gfCNCPoint2[9660] = {X 255.0630, Y 50.0697, Z -3.0000, A 0.000, B 0.000, C 0.000 }
gfCNCPoint2[9661] = {X 254.3405, Y 49.1989, Z -3.0000, A 0.000, B 0.000, C 0.000 }
gfCNCPoint2[9662] = {X 253.7617, Y 48.2267, Z -3.0000, A 0.000, B 0.000, C 0.000 }
gfCNCPoint2[9663] = {X 253.3406, Y 47.1766, Z -3.0000, A 0.000, B 0.000, C 0.000 }
gfCNCPoint2[9664] = {X 252.9194, Y 48.2267, Z -3.0000, A 0.000, B 0.000, C 0.000 }
gfCNCPoint2[9665] = {X 252.3406, Y 49.1989, Z -3.0000, A 0.000, B 0.000, C 0.000 }
gfCNCPoint2[9666] = {X 251.6182, Y 50.0697, Z -3.0000, A 0.000, B 0.000, C 0.000 }
gfCNCPoint2[9667] = {X 251.5688, Y 50.1201, Z -3.0000, A 0.000, B 0.000, C 0.000 }
gfCNCPoint2[9668] = {X 251.5189, Y 50.1700, Z -3.0000, A 0.000, B 0.000, C 0.000 }
gfCNCPoint2[9669] = {X 250.7133, Y 50.8599, Z -3.0000, A 0.000, B 0.000, C 0.000 }
gfCNCPoint2[9670] = {X 249.8160, Y 51.4254, Z -3.0000, A 0.000, B 0.000, C 0.000 }
gfCNCPoint2[9671] = {X 248.8461, Y 51.8545, Z -3.0000, A 0.000, B 0.000, C 0.000 }
gfCNCPoint2[9672] = {X 247.8241, Y 52.1381, Z -3.0000, A 0.000, B 0.000, C 0.000 }
gfCNCPoint2[9673] = {X 247.8929, Y 52.2639, Z -3.0000, A 0.000, B 0.000, C 0.000 }
gfCNCPoint2[9674] = {X 247.9603, Y 52.3905, Z -3.0000, A 0.000, B 0.000, C 0.000 }
gfCNCPoint2[9675] = {X 250.3409, Y 53.3186, Z -3.0000, A 0.000, B 0.000, C 0.000 }
gfCNCPoint2[9676] = {X 264.1528, Y 58.7989, Z -3.0000, A 0.000, B 0.000, C 0.000 }
gfCNCPoint2[9677] = {X 264.1527, Y 58.0000, Z -3.0000, A 0.000, B 0.000, C 0.000 }
gfCNCPoint2[9678] = {X 264.2034, Y 56.8945, Z -3.0000, A 0.000, B 0.000, C 0.000 }
gfCNCPoint2[9679] = {X 264.3550, Y 55.7982, Z -3.0000, A 0.000, B 0.000, C 0.000 }
gfCNCPoint2[9680] = {X 264.4114, Y 55.5135, Z -3.0000, A 0.000, B 0.000, C 0.000 }
gfCNCPoint2[9681] = {X 264.4745, Y 55.2303, Z -3.0000, A 0.000, B 0.000, C 0.000 }
gfCNCPoint2[9682] = {X 264.9369, Y 53.7185, Z -3.0000, A 0.000, B 0.000, C 0.000 }
gfCNCPoint2[9683] = {X 265.5928, Y 52.2800, Z -3.0000, A 0.000, B 0.000, C 0.000 }
gfCNCPoint2[9684] = {X 262.1384, Y 52.2800, Z -3.0000, A 0.000, B 0.000, C 0.000 }
gfCNCPoint2[9685] = {X 262.1384, Y 49.8800, Z -3.0000, A 0.000, B 0.000, C 0.000 }
gfCNCPoint2[9686] = {X 260.2876, Y 49.8800, Z -3.0000, A 0.000, B 0.000, C 0.000 }
gfCNCPoint2[9687] = {X 259.2646, Y 49.7716, Z -3.0000, A 0.000, B 0.000, C 0.000 }
gfCNCPoint2[9688] = {X 258.2870, Y 49.4511, Z -3.0000, A 0.000, B 0.000, C 0.000 }
gfCNCPoint2[9689] = {X 257.3984, Y 48.9328, Z -3.0000, A 0.000, B 0.000, C 0.000 }
gfCNCPoint2[9690] = {X 256.6382, Y 48.2398, Z -3.0000, A 0.000, B 0.000, C 0.000 }
gfCNCPoint2[9691] = {X 256.0401, Y 47.4028, Z -3.0000, A 0.000, B 0.000, C 0.000 }
gfCNCPoint2[9692] = {X 255.6308, Y 46.4590, Z -3.0000, A 0.000, B 0.000, C 0.000 }
gfCNCPoint2[9693] = {X 255.4666, Y 45.7568, Z -3.0000, A 0.000, B 0.000, C 0.000 }
gfCNCPoint2[9694] = {X 255.4077, Y 45.0380, Z -3.0000, A 0.000, B 0.000, C 0.000 }
gfCNCPoint2[9695] = {X 255.4080, Y 44.1416, Z -3.0000, A 0.000, B 0.000, C 0.000 }
gfCNCPoint2[9696] = {X 255.5183, Y 43.1751, Z -3.0000, A 0.000, B 0.000, C 0.000 }
gfCNCPoint2[9697] = {X 255.8181, Y 42.2496, Z -3.0000, A 0.000, B 0.000, C 0.000 }
gfCNCPoint2[9698] = {X 256.2955, Y 41.4020, Z -3.0000, A 0.000, B 0.000, C 0.000 }
gfCNCPoint2[9699] = {X 256.9315, Y 40.6660, Z -3.0000, A 0.000, B 0.000, C 0.000 }
gfCNCPoint2[9700] = {X 256.9315, Y 35.0338, Z -3.0000, A 0.000, B 0.000, C 0.000 }
gfCNCPoint2[9701] = {X 255.1091, Y 35.0338, Z -3.0000, A 0.000, B 0.000, C 0.000 }
gfCNCPoint2[9702] = {X 251.0864, Y 42.8703, Z -3.0000, A 0.000, B 0.000, C 0.000 }
gfCNCPoint2[9703] = {X 251.2236, Y 43.5126, Z -3.0000, A 0.000, B 0.000, C 0.000 }
gfCNCPoint2[9704] = {X 251.2734, Y 44.1675, Z -3.0000, A 0.000, B 0.000, C 0.000 }
gfCNCPoint2[9705] = {X 251.2736, Y 45.0000, Z -3.0000, A 0.000, B 0.000, C 0.000 }
gfCNCPoint2[9706] = {X 251.2174, Y 45.7380, Z -3.0000, A 0.000, B 0.000, C 0.000 }
gfCNCPoint2[9707] = {X 251.0503, Y 46.4590, Z -3.0000, A 0.000, B 0.000, C 0.000 }
gfCNCPoint2[9708] = {X 250.6346, Y 47.4142, Z -3.0000, A 0.000, B 0.000, C 0.000 }
gfCNCPoint2[9709] = {X 250.0255, Y 48.2593, Z -3.0000, A 0.000, B 0.000, C 0.000 }
gfCNCPoint2[9710] = {X 249.2510, Y 48.9560, Z -3.0000, A 0.000, B 0.000, C 0.000 }
gfCNCPoint2[9711] = {X 248.3462, Y 49.4723, Z -3.0000, A 0.000, B 0.000, C 0.000 }
gfCNCPoint2[9712] = {X 247.3525, Y 49.7849, Z -3.0000, A 0.000, B 0.000, C 0.000 }
gfCNCPoint2[9713] = {X 246.8754, Y 49.8562, Z -3.0000, A 0.000, B 0.000, C 0.000 }
gfCNCPoint2[9714] = {X 246.3936, Y 49.8800, Z -3.0000, A 0.000, B 0.000, C 0.000 }
gfCNCPoint2[9715] = {X 242.5312, Y 49.8800, Z -3.0000, A 0.000, B 0.000, C 0.000 }
gfCNCPoint2[9716] = {X 242.5312, Y 49.4000, Z -3.0000, A 0.000, B 0.000, C 0.000 }
gfCNCPoint2[9717] = {X 239.8075, Y 49.4000, Z -3.0000, A 0.000, B 0.000, C 0.000 }
gfCNCPoint2[9718] = {X 238.8284, Y 49.2897, Z -3.0000, A 0.000, B 0.000, C 0.000 }
gfCNCPoint2[9719] = {X 237.8984, Y 48.9643, Z -3.0000, A 0.000, B 0.000, C 0.000 }
gfCNCPoint2[9720] = {X 237.0641, Y 48.4401, Z -3.0000, A 0.000, B 0.000, C 0.000 }
gfCNCPoint2[9721] = {X 236.3674, Y 47.7434, Z -3.0000, A 0.000, B 0.000, C 0.000 }
gfCNCPoint2[9722] = {X 235.8432, Y 46.9091, Z -3.0000, A 0.000, B 0.000, C 0.000 }
gfCNCPoint2[9723] = {X 235.5178, Y 45.9791, Z -3.0000, A 0.000, B 0.000, C 0.000 }
gfCNCPoint2[9724] = {X 235.4075, Y 45.0000, Z -3.0000, A 0.000, B 0.000, C 0.000 }
gfCNCPoint2[9725] = {X 235.4079, Y 44.1483, Z -3.0000, A 0.000, B 0.000, C 0.000 }
gfCNCPoint2[9726] = {X 235.5063, Y 43.2816, Z -3.0000, A 0.000, B 0.000, C 0.000 }
gfCNCPoint2[9727] = {X 235.7737, Y 42.4514, Z -3.0000, A 0.000, B 0.000, C 0.000 }
gfCNCPoint2[9728] = {X 236.1996, Y 41.6903, Z -3.0000, A 0.000, B 0.000, C 0.000 }
gfCNCPoint2[9729] = {X 236.7672, Y 41.0281, Z -3.0000, A 0.000, B 0.000, C 0.000 }
gfCNCPoint2[9730] = {X 237.4544, Y 40.4909, Z -3.0000, A 0.000, B 0.000, C 0.000 }
gfCNCPoint2[9731] = {X 238.2339, Y 40.0998, Z -3.0000, A 0.000, B 0.000, C 0.000 }
gfCNCPoint2[9732] = {X 242.1750, Y 32.3856, Z -3.0000, A 0.000, B 0.000, C 0.000 }
gfCNCPoint2[9733] = {X 241.0115, Y 31.5932, Z -3.0000, A 0.000, B 0.000, C 0.000 }
gfCNCPoint2[9734] = {X 239.9546, Y 30.6635, Z -3.0000, A 0.000, B 0.000, C 0.000 }
gfCNCPoint2[9735] = {X 239.0203, Y 29.6105, Z -3.0000, A 0.000, B 0.000, C 0.000 }
gfCNCPoint2[9736] = {X 238.2230, Y 28.4504, Z -3.0000, A 0.000, B 0.000, C 0.000 }
gfCNCPoint2[9737] = {X 237.5748, Y 27.2009, Z -3.0000, A 0.000, B 0.000, C 0.000 }
gfCNCPoint2[9738] = {X 237.0856, Y 25.8809, Z -3.0000, A 0.000, B 0.000, C 0.000 }
gfCNCPoint2[9739] = {X 236.6638, Y 24.0613, Z -3.0000, A 0.000, B 0.000, C 0.000 }
gfCNCPoint2[9740] = {X 236.4490, Y 22.2058, Z -3.0000, A 0.000, B 0.000, C 0.000 }
gfCNCPoint2[9741] = {X 236.4438, Y 20.3378, Z -3.0000, A 0.000, B 0.000, C 0.000 }
gfCNCPoint2[9742] = {X 236.6483, Y 18.4812, Z -3.0000, A 0.000, B 0.000, C 0.000 }
gfCNCPoint2[9743] = {X 237.0599, Y 16.6592, Z -3.0000, A 0.000, B 0.000, C 0.000 }
gfCNCPoint2[9744] = {X 237.6340, Y 15.0730, Z -3.0000, A 0.000, B 0.000, C 0.000 }
gfCNCPoint2[9745] = {X 238.4262, Y 13.5836, Z -3.0000, A 0.000, B 0.000, C 0.000 }
gfCNCPoint2[9746] = {X 239.4206, Y 12.2210, Z -3.0000, A 0.000, B 0.000, C 0.000 }
gfCNCPoint2[9747] = {X 240.5972, Y 11.0123, Z -3.0000, A 0.000, B 0.000, C 0.000 }
gfCNCPoint2[9748] = {X 241.9327, Y 9.9816, Z -3.0000, A 0.000, B 0.000, C 0.000 }
gfCNCPoint2[9749] = {X 243.4002, Y 9.1497, Z -3.0000, A 0.000, B 0.000, C 0.000 }
gfCNCPoint2[9750] = {X 244.9704, Y 8.5332, Z -3.0000, A 0.000, B 0.000, C 0.000 }
gfCNCPoint2[9751] = {X 246.6119, Y 8.1444, Z -3.0000, A 0.000, B 0.000, C 0.000 }
gfCNCPoint2[9752] = {X 248.7155, Y 7.8721, Z -3.0000, A 0.000, B 0.000, C 0.000 }
gfCNCPoint2[9753] = {X 250.8351, Y 7.7912, Z -3.0000, A 0.000, B 0.000, C 0.000 }
gfCNCPoint2[9754] = {X 266.7640, Y 7.7912, Z -3.0000, A 0.000, B 0.000, C 0.000 }
gfCNCPoint2[9755] = {X 267.7368, Y 7.9081, Z -3.0000, A 0.000, B 0.000, C 0.000 }
gfCNCPoint2[9756] = {X 268.6596, Y 8.2373, Z -3.0000, A 0.000, B 0.000, C 0.000 }
gfCNCPoint2[9757] = {X 269.4868, Y 8.7623, Z -3.0000, A 0.000, B 0.000, C 0.000 }
gfCNCPoint2[9758] = {X 270.1773, Y 9.4573, Z -3.0000, A 0.000, B 0.000, C 0.000 }
gfCNCPoint2[9759] = {X 270.6971, Y 10.2878, Z -3.0000, A 0.000, B 0.000, C 0.000 }
gfCNCPoint2[9760] = {X 271.0203, Y 11.2127, Z -3.0000, A 0.000, B 0.000, C 0.000 }
gfCNCPoint2[9761] = {X 271.1310, Y 12.1862, Z -3.0000, A 0.000, B 0.000, C 0.000 }
gfCNCPoint2[9762] = {X 271.1308, Y 13.0233, Z -3.0000, A 0.000, B 0.000, C 0.000 }
gfCNCPoint2[9763] = {X 271.0225, Y 13.9494, Z -3.0000, A 0.000, B 0.000, C 0.000 }
gfCNCPoint2[9764] = {X 270.7215, Y 14.8318, Z -3.0000, A 0.000, B 0.000, C 0.000 }
gfCNCPoint2[9765] = {X 270.2413, Y 15.6310, Z -3.0000, A 0.000, B 0.000, C 0.000 }
gfCNCPoint2[9766] = {X 269.6034, Y 16.3111, Z -3.0000, A 0.000, B 0.000, C 0.000 }
gfCNCPoint2[9767] = {X 269.6032, Y 40.8756, Z -3.0000, A 0.000, B 0.000, C 0.000 }
gfCNCPoint2[9768] = {X 270.2480, Y 41.5647, Z -3.0000, A 0.000, B 0.000, C 0.000 }
gfCNCPoint2[9769] = {X 270.7309, Y 42.3755, Z -3.0000, A 0.000, B 0.000, C 0.000 }
gfCNCPoint2[9770] = {X 271.0299, Y 43.2706, Z -3.0000, A 0.000, B 0.000, C 0.000 }
gfCNCPoint2[9771] = {X 271.1310, Y 44.2089, Z -3.0000, A 0.000, B 0.000, C 0.000 }
gfCNCPoint2[9772] = {X 271.1310, Y 45.0000, Z -3.0000, A 0.000, B 0.000, C 0.000 }
gfCNCPoint2[9773] = {X 271.0207, Y 45.9791, Z -3.0000, A 0.000, B 0.000, C 0.000 }
gfCNCPoint2[9774] = {X 270.6953, Y 46.9091, Z -3.0000, A 0.000, B 0.000, C 0.000 }
gfCNCPoint2[9775] = {X 270.1711, Y 47.7434, Z -3.0000, A 0.000, B 0.000, C 0.000 }
gfCNCPoint2[9776] = {X 269.4744, Y 48.4401, Z -3.0000, A 0.000, B 0.000, C 0.000 }
gfCNCPoint2[9777] = {X 268.6401, Y 48.9643, Z -3.0000, A 0.000, B 0.000, C 0.000 }
gfCNCPoint2[9778] = {X 267.7101, Y 49.2897, Z -3.0000, A 0.000, B 0.000, C 0.000 }
gfCNCPoint2[9779] = {X 266.7310, Y 49.4000, Z -3.0000, A 0.000, B 0.000, C 0.000 }
gfCNCPoint2[9780] = {X 260.2876, Y 49.4000, Z -3.0000, A 0.000, B 0.000, C 0.000 }
gfCNCPoint2[9781] = {X 259.3085, Y 49.2897, Z -3.0000, A 0.000, B 0.000, C 0.000 }
gfCNCPoint2[9782] = {X 258.3785, Y 48.9643, Z -3.0000, A 0.000, B 0.000, C 0.000 }
gfCNCPoint2[9783] = {X 257.5442, Y 48.4400, Z -3.0000, A 0.000, B 0.000, C 0.000 }
gfCNCPoint2[9784] = {X 256.8475, Y 47.7433, Z -3.0000, A 0.000, B 0.000, C 0.000 }
gfCNCPoint2[9785] = {X 256.3233, Y 46.9091, Z -3.0000, A 0.000, B 0.000, C 0.000 }
gfCNCPoint2[9786] = {X 255.9979, Y 45.9791, Z -3.0000, A 0.000, B 0.000, C 0.000 }
gfCNCPoint2[9787] = {X 255.8876, Y 45.0000, Z -3.0000, A 0.000, B 0.000, C 0.000 }
gfCNCPoint2[9788] = {X 255.8880, Y 44.1483, Z -3.0000, A 0.000, B 0.000, C 0.000 }
gfCNCPoint2[9789] = {X 255.9984, Y 43.2275, Z -3.0000, A 0.000, B 0.000, C 0.000 }
gfCNCPoint2[9790] = {X 256.2993, Y 42.3503, Z -3.0000, A 0.000, B 0.000, C 0.000 }
gfCNCPoint2[9791] = {X 256.7775, Y 41.5556, Z -3.0000, A 0.000, B 0.000, C 0.000 }
gfCNCPoint2[9792] = {X 257.4115, Y 40.8789, Z -3.0000, A 0.000, B 0.000, C 0.000 }
gfCNCPoint2[9793] = {X 257.4115, Y 34.5538, Z -3.0000, A 0.000, B 0.000, C 0.000 }
gfCNCPoint2[9794] = {X 254.8159, Y 34.5538, Z -3.0000, A 0.000, B 0.000, C 0.000 }
gfCNCPoint2[9795] = {X 250.5702, Y 42.8248, Z -3.0000, A 0.000, B 0.000, C 0.000 }
gfCNCPoint2[9796] = {X 250.7374, Y 43.5079, Z -3.0000, A 0.000, B 0.000, C 0.000 }
gfCNCPoint2[9797] = {X 250.7936, Y 44.2089, Z -3.0000, A 0.000, B 0.000, C 0.000 }
gfCNCPoint2[9798] = {X 250.7936, Y 45.0000, Z -3.0000, A 0.000, B 0.000, C 0.000 }
gfCNCPoint2[9799] = {X 250.6832, Y 45.9791, Z -3.0000, A 0.000, B 0.000, C 0.000 }
gfCNCPoint2[9800] = {X 250.3578, Y 46.9091, Z -3.0000, A 0.000, B 0.000, C 0.000 }
gfCNCPoint2[9801] = {X 249.8336, Y 47.7434, Z -3.0000, A 0.000, B 0.000, C 0.000 }
gfCNCPoint2[9802] = {X 249.1369, Y 48.4401, Z -3.0000, A 0.000, B 0.000, C 0.000 }
gfCNCPoint2[9803] = {X 248.3026, Y 48.9643, Z -3.0000, A 0.000, B 0.000, C 0.000 }
gfCNCPoint2[9804] = {X 247.3727, Y 49.2897, Z -3.0000, A 0.000, B 0.000, C 0.000 }
gfCNCPoint2[9805] = {X 246.3936, Y 49.4000, Z -3.0000, A 0.000, B 0.000, C 0.000 }
gfCNCPoint2[9806] = {X 242.5312, Y 49.4000, Z -3.0000, A 0.000, B 0.000, C 0.000 }
gfCNCPoint2[9807] = {X 242.5312, Y 49.8800, Z -3.0000, A 0.000, B 0.000, C 0.000 }
gfCNCPoint2[9808] = {X 243.4812, Y 50.5824, Z -3.0000, A 0.000, B 0.000, C 0.000 }
gfCNCPoint2[9809] = {X 244.3384, Y 51.3953, Z -3.0000, A 0.000, B 0.000, C 0.000 }
gfCNCPoint2[9810] = {X 245.0903, Y 52.3066, Z -3.0000, A 0.000, B 0.000, C 0.000 }
gfCNCPoint2[9811] = {X 245.7256, Y 53.3027, Z -3.0000, A 0.000, B 0.000, C 0.000 }
gfCNCPoint2[9812] = {X 245.9756, Y 53.7844, Z -3.0000, A 0.000, B 0.000, C 0.000 }
gfCNCPoint2[9813] = {X 246.1981, Y 54.2794, Z -3.0000, A 0.000, B 0.000, C 0.000 }
gfCNCPoint2[9814] = {X 249.4592, Y 55.5508, Z -3.0000, A 0.000, B 0.000, C 0.000 }
gfCNCPoint2[9815] = {X 267.2831, Y 62.6229, Z -3.0000, A 0.000, B 0.000, C 0.000 }
gfCNCPoint2[9816] = {X 266.8847, Y 61.4476, Z -3.0000, A 0.000, B 0.000, C 0.000 }
gfCNCPoint2[9817] = {X 266.6400, Y 60.2310, Z -3.0000, A 0.000, B 0.000, C 0.000 }
gfCNCPoint2[9818] = {X 266.5529, Y 58.9930, Z -3.0000, A 0.000, B 0.000, C 0.000 }
gfCNCPoint2[9819] = {X 266.5527, Y 58.0000, Z -3.0000, A 0.000, B 0.000, C 0.000 }
gfCNCPoint2[9820] = {X 266.6262, Y 56.8093, Z -3.0000, A 0.000, B 0.000, C 0.000 }
gfCNCPoint2[9821] = {X 266.8456, Y 55.6367, Z -3.0000, A 0.000, B 0.000, C 0.000 }
gfCNCPoint2[9822] = {X 267.2076, Y 54.5000, Z -3.0000, A 0.000, B 0.000, C 0.000 }
gfCNCPoint2[9823] = {X 267.7067, Y 53.4164, Z -3.0000, A 0.000, B 0.000, C 0.000 }
gfCNCPoint2[9824] = {X 268.4728, Y 52.2132, Z -3.0000, A 0.000, B 0.000, C 0.000 }
gfCNCPoint2[9825] = {X 269.4075, Y 51.1357, Z -3.0000, A 0.000, B 0.000, C 0.000 }
gfCNCPoint2[9826] = {X 270.4903, Y 50.2072, Z -3.0000, A 0.000, B 0.000, C 0.000 }
gfCNCPoint2[9827] = {X 271.6979, Y 49.4479, Z -3.0000, A 0.000, B 0.000, C 0.000 }
gfCNCPoint2[9828] = {X 273.0039, Y 48.8744, Z -3.0000, A 0.000, B 0.000, C 0.000 }
gfCNCPoint2[9829] = {X 274.3800, Y 48.4989, Z -3.0000, A 0.000, B 0.000, C 0.000 }
gfCNCPoint2[9830] = {X 275.3020, Y 48.3648, Z -3.0000, A 0.000, B 0.000, C 0.000 }
gfCNCPoint2[9831] = {X 276.2327, Y 48.3200, Z -3.0000, A 0.000, B 0.000, C 0.000 }
gfCNCPoint2[9832] = {X 281.0411, Y 48.3200, Z -3.0000, A 0.000, B 0.000, C 0.000 }
gfCNCPoint2[9833] = {X 280.4347, Y 47.5134, Z -3.0000, A 0.000, B 0.000, C 0.000 }
gfCNCPoint2[9834] = {X 280.0072, Y 46.5992, Z -3.0000, A 0.000, B 0.000, C 0.000 }
gfCNCPoint2[9835] = {X 279.7768, Y 45.6167, Z -3.0000, A 0.000, B 0.000, C 0.000 }
gfCNCPoint2[9836] = {X 279.7488, Y 45.3288, Z -3.0000, A 0.000, B 0.000, C 0.000 }
gfCNCPoint2[9837] = {X 279.7378, Y 45.0398, Z -3.0000, A 0.000, B 0.000, C 0.000 }
gfCNCPoint2[9838] = {X 279.7377, Y 44.2039, Z -3.0000, A 0.000, B 0.000, C 0.000 }
gfCNCPoint2[9839] = {X 279.8424, Y 43.2205, Z -3.0000, A 0.000, B 0.000, C 0.000 }
gfCNCPoint2[9840] = {X 280.1412, Y 42.2777, Z -3.0000, A 0.000, B 0.000, C 0.000 }
gfCNCPoint2[9841] = {X 280.6222, Y 41.4136, Z -3.0000, A 0.000, B 0.000, C 0.000 }
gfCNCPoint2[9842] = {X 281.2659, Y 40.6627, Z -3.0000, A 0.000, B 0.000, C 0.000 }
gfCNCPoint2[9843] = {X 281.2655, Y 16.5245, Z -3.0000, A 0.000, B 0.000, C 0.000 }
gfCNCPoint2[9844] = {X 280.6242, Y 15.7828, Z -3.0000, A 0.000, B 0.000, C 0.000 }
gfCNCPoint2[9845] = {X 280.1442, Y 14.9280, Z -3.0000, A 0.000, B 0.000, C 0.000 }
gfCNCPoint2[9846] = {X 279.8447, Y 13.9944, Z -3.0000, A 0.000, B 0.000, C 0.000 }
gfCNCPoint2[9847] = {X 279.7378, Y 13.0198, Z -3.0000, A 0.000, B 0.000, C 0.000 }
gfCNCPoint2[9848] = {X 279.7377, Y 12.1868, Z -3.0000, A 0.000, B 0.000, C 0.000 }
gfCNCPoint2[9849] = {X 279.8242, Y 11.2717, Z -3.0000, A 0.000, B 0.000, C 0.000 }
gfCNCPoint2[9850] = {X 280.0808, Y 10.3891, Z -3.0000, A 0.000, B 0.000, C 0.000 }
gfCNCPoint2[9851] = {X 280.5256, Y 9.5281, Z -3.0000, A 0.000, B 0.000, C 0.000 }
gfCNCPoint2[9852] = {X 281.1317, Y 8.7718, Z -3.0000, A 0.000, B 0.000, C 0.000 }
gfCNCPoint2[9853] = {X 281.8752, Y 8.1503, Z -3.0000, A 0.000, B 0.000, C 0.000 }
gfCNCPoint2[9854] = {X 282.7270, Y 7.6880, Z -3.0000, A 0.000, B 0.000, C 0.000 }
gfCNCPoint2[9855] = {X 283.6533, Y 7.4030, Z -3.0000, A 0.000, B 0.000, C 0.000 }
gfCNCPoint2[9856] = {X 284.6177, Y 7.3068, Z -3.0000, A 0.000, B 0.000, C 0.000 }
gfCNCPoint2[9857] = {X 291.0611, Y 7.3068, Z -3.0000, A 0.000, B 0.000, C 0.000 }
gfCNCPoint2[9858] = {X 292.0255, Y 7.4030, Z -3.0000, A 0.000, B 0.000, C 0.000 }
gfCNCPoint2[9859] = {X 292.9518, Y 7.6880, Z -3.0000, A 0.000, B 0.000, C 0.000 }
gfCNCPoint2[9860] = {X 293.8036, Y 8.1503, Z -3.0000, A 0.000, B 0.000, C 0.000 }
gfCNCPoint2[9861] = {X 294.5471, Y 8.7718, Z -3.0000, A 0.000, B 0.000, C 0.000 }
gfCNCPoint2[9862] = {X 295.1533, Y 9.5281, Z -3.0000, A 0.000, B 0.000, C 0.000 }
gfCNCPoint2[9863] = {X 295.5980, Y 10.3891, Z -3.0000, A 0.000, B 0.000, C 0.000 }
gfCNCPoint2[9864] = {X 295.8044, Y 11.0397, Z -3.0000, A 0.000, B 0.000, C 0.000 }
gfCNCPoint2[9865] = {X 295.9180, Y 11.7127, Z -3.0000, A 0.000, B 0.000, C 0.000 }
gfCNCPoint2[9866] = {X 295.9354, Y 11.9495, Z -3.0000, A 0.000, B 0.000, C 0.000 }
gfCNCPoint2[9867] = {X 295.9411, Y 12.1868, Z -3.0000, A 0.000, B 0.000, C 0.000 }
gfCNCPoint2[9868] = {X 295.9409, Y 13.0237, Z -3.0000, A 0.000, B 0.000, C 0.000 }
gfCNCPoint2[9869] = {X 295.9342, Y 13.2382, Z -3.0000, A 0.000, B 0.000, C 0.000 }
gfCNCPoint2[9870] = {X 295.9180, Y 13.4521, Z -3.0000, A 0.000, B 0.000, C 0.000 }
gfCNCPoint2[9871] = {X 298.3067, Y 13.6853, Z -3.0000, A 0.000, B 0.000, C 0.000 }
gfCNCPoint2[9872] = {X 298.1360, Y 14.6938, Z -3.0000, A 0.000, B 0.000, C 0.000 }
gfCNCPoint2[9873] = {X 297.8257, Y 15.6685, Z -3.0000, A 0.000, B 0.000, C 0.000 }
gfCNCPoint2[9874] = {X 297.3819, Y 16.5900, Z -3.0000, A 0.000, B 0.000, C 0.000 }
gfCNCPoint2[9875] = {X 296.8132, Y 17.4403, Z -3.0000, A 0.000, B 0.000, C 0.000 }
gfCNCPoint2[9876] = {X 296.8136, Y 19.2365, Z -3.0000, A 0.000, B 0.000, C 0.000 }
gfCNCPoint2[9877] = {X 299.7997, Y 19.2365, Z -3.0000, A 0.000, B 0.000, C 0.000 }
gfCNCPoint2[9878] = {X 299.7999, Y 17.4399, Z -3.0000, A 0.000, B 0.000, C 0.000 }
gfCNCPoint2[9879] = {X 299.2314, Y 16.5898, Z -3.0000, A 0.000, B 0.000, C 0.000 }
gfCNCPoint2[9880] = {X 298.7876, Y 15.6683, Z -3.0000, A 0.000, B 0.000, C 0.000 }
gfCNCPoint2[9881] = {X 298.4773, Y 14.6937, Z -3.0000, A 0.000, B 0.000, C 0.000 }
gfCNCPoint2[9882] = {X 298.3067, Y 13.6853, Z -3.0000, A 0.000, B 0.000, C 0.000 }
gfCNCPoint2[9883] = {X 295.9180, Y 13.4521, Z -3.0000, A 0.000, B 0.000, C 0.000 }
gfCNCPoint2[9884] = {X 295.7559, Y 14.3097, Z -3.0000, A 0.000, B 0.000, C 0.000 }
gfCNCPoint2[9885] = {X 295.4436, Y 15.1246, Z -3.0000, A 0.000, B 0.000, C 0.000 }
gfCNCPoint2[9886] = {X 294.9912, Y 15.8710, Z -3.0000, A 0.000, B 0.000, C 0.000 }
gfCNCPoint2[9887] = {X 294.4130, Y 16.5247, Z -3.0000, A 0.000, B 0.000, C 0.000 }
gfCNCPoint2[9888] = {X 294.4141, Y 21.6365, Z -3.0000, A 0.000, B 0.000, C 0.000 }
gfCNCPoint2[9889] = {X 302.1995, Y 21.6365, Z -3.0000, A 0.000, B 0.000, C 0.000 }
gfCNCPoint2[9890] = {X 302.2000, Y 16.5244, Z -3.0000, A 0.000, B 0.000, C 0.000 }
gfCNCPoint2[9891] = {X 301.6220, Y 15.8706, Z -3.0000, A 0.000, B 0.000, C 0.000 }
gfCNCPoint2[9892] = {X 301.1696, Y 15.1244, Z -3.0000, A 0.000, B 0.000, C 0.000 }
gfCNCPoint2[9893] = {X 300.8574, Y 14.3095, Z -3.0000, A 0.000, B 0.000, C 0.000 }
gfCNCPoint2[9894] = {X 300.6953, Y 13.4521, Z -3.0000, A 0.000, B 0.000, C 0.000 }
gfCNCPoint2[9895] = {X 300.6791, Y 13.2371, Z -3.0000, A 0.000, B 0.000, C 0.000 }
gfCNCPoint2[9896] = {X 300.6724, Y 13.0215, Z -3.0000, A 0.000, B 0.000, C 0.000 }
gfCNCPoint2[9897] = {X 300.6723, Y 12.1868, Z -3.0000, A 0.000, B 0.000, C 0.000 }
gfCNCPoint2[9898] = {X 300.6780, Y 11.9495, Z -3.0000, A 0.000, B 0.000, C 0.000 }
gfCNCPoint2[9899] = {X 300.6953, Y 11.7127, Z -3.0000, A 0.000, B 0.000, C 0.000 }
gfCNCPoint2[9900] = {X 300.8090, Y 11.0397, Z -3.0000, A 0.000, B 0.000, C 0.000 }
gfCNCPoint2[9901] = {X 301.0154, Y 10.3891, Z -3.0000, A 0.000, B 0.000, C 0.000 }
gfCNCPoint2[9902] = {X 301.4601, Y 9.5281, Z -3.0000, A 0.000, B 0.000, C 0.000 }
gfCNCPoint2[9903] = {X 302.0662, Y 8.7718, Z -3.0000, A 0.000, B 0.000, C 0.000 }
gfCNCPoint2[9904] = {X 302.8098, Y 8.1503, Z -3.0000, A 0.000, B 0.000, C 0.000 }
gfCNCPoint2[9905] = {X 303.6616, Y 7.6880, Z -3.0000, A 0.000, B 0.000, C 0.000 }
gfCNCPoint2[9906] = {X 304.5879, Y 7.4030, Z -3.0000, A 0.000, B 0.000, C 0.000 }
gfCNCPoint2[9907] = {X 305.5523, Y 7.3068, Z -3.0000, A 0.000, B 0.000, C 0.000 }
gfCNCPoint2[9908] = {X 311.9957, Y 7.3068, Z -3.0000, A 0.000, B 0.000, C 0.000 }
gfCNCPoint2[9909] = {X 312.9478, Y 7.4006, Z -3.0000, A 0.000, B 0.000, C 0.000 }
gfCNCPoint2[9910] = {X 313.8632, Y 7.6783, Z -3.0000, A 0.000, B 0.000, C 0.000 }
gfCNCPoint2[9911] = {X 314.7069, Y 8.1292, Z -3.0000, A 0.000, B 0.000, C 0.000 }
gfCNCPoint2[9912] = {X 315.4464, Y 8.7361, Z -3.0000, A 0.000, B 0.000, C 0.000 }
gfCNCPoint2[9913] = {X 316.0533, Y 9.4756, Z -3.0000, A 0.000, B 0.000, C 0.000 }
gfCNCPoint2[9914] = {X 316.5043, Y 10.3193, Z -3.0000, A 0.000, B 0.000, C 0.000 }
gfCNCPoint2[9915] = {X 316.7820, Y 11.2348, Z -3.0000, A 0.000, B 0.000, C 0.000 }
gfCNCPoint2[9916] = {X 316.8757, Y 12.1868, Z -3.0000, A 0.000, B 0.000, C 0.000 }
gfCNCPoint2[9917] = {X 316.8755, Y 13.0237, Z -3.0000, A 0.000, B 0.000, C 0.000 }
gfCNCPoint2[9918] = {X 316.7681, Y 13.9973, Z -3.0000, A 0.000, B 0.000, C 0.000 }
gfCNCPoint2[9919] = {X 316.4684, Y 14.9299, Z -3.0000, A 0.000, B 0.000, C 0.000 }
gfCNCPoint2[9920] = {X 315.9885, Y 15.7838, Z -3.0000, A 0.000, B 0.000, C 0.000 }
gfCNCPoint2[9921] = {X 315.3477, Y 16.5246, Z -3.0000, A 0.000, B 0.000, C 0.000 }
gfCNCPoint2[9922] = {X 315.3475, Y 40.6620, Z -3.0000, A 0.000, B 0.000, C 0.000 }
gfCNCPoint2[9923] = {X 315.9888, Y 41.4035, Z -3.0000, A 0.000, B 0.000, C 0.000 }
gfCNCPoint2[9924] = {X 316.4690, Y 42.2583, Z -3.0000, A 0.000, B 0.000, C 0.000 }
gfCNCPoint2[9925] = {X 316.7686, Y 43.1918, Z -3.0000, A 0.000, B 0.000, C 0.000 }
gfCNCPoint2[9926] = {X 316.8755, Y 44.1664, Z -3.0000, A 0.000, B 0.000, C 0.000 }
gfCNCPoint2[9927] = {X 316.8757, Y 45.0000, Z -3.0000, A 0.000, B 0.000, C 0.000 }
gfCNCPoint2[9928] = {X 316.8749, Y 45.0899, Z -3.0000, A 0.000, B 0.000, C 0.000 }
gfCNCPoint2[9929] = {X 316.8724, Y 45.1799, Z -3.0000, A 0.000, B 0.000, C 0.000 }
gfCNCPoint2[9930] = {X 316.8594, Y 45.3987, Z -3.0000, A 0.000, B 0.000, C 0.000 }
gfCNCPoint2[9931] = {X 316.8366, Y 45.6167, Z -3.0000, A 0.000, B 0.000, C 0.000 }
gfCNCPoint2[9932] = {X 316.6062, Y 46.5992, Z -3.0000, A 0.000, B 0.000, C 0.000 }
gfCNCPoint2[9933] = {X 316.1787, Y 47.5134, Z -3.0000, A 0.000, B 0.000, C 0.000 }
gfCNCPoint2[9934] = {X 315.5723, Y 48.3200, Z -3.0000, A 0.000, B 0.000, C 0.000 }
gfCNCPoint2[9935] = {X 315.2205, Y 47.9934, Z -3.0000, A 0.000, B 0.000, C 0.000 }
gfCNCPoint2[9936] = {X 314.5413, Y 48.5889, Z -3.0000, A 0.000, B 0.000, C 0.000 }
gfCNCPoint2[9937] = {X 313.7548, Y 49.0331, Z -3.0000, A 0.000, B 0.000, C 0.000 }
gfCNCPoint2[9938] = {X 312.8942, Y 49.3073, Z -3.0000, A 0.000, B 0.000, C 0.000 }
gfCNCPoint2[9939] = {X 311.9957, Y 49.4000, Z -3.0000, A 0.000, B 0.000, C 0.000 }
gfCNCPoint2[9940] = {X 305.5523, Y 49.4000, Z -3.0000, A 0.000, B 0.000, C 0.000 }
gfCNCPoint2[9941] = {X 304.5732, Y 49.2897, Z -3.0000, A 0.000, B 0.000, C 0.000 }
gfCNCPoint2[9942] = {X 303.6432, Y 48.9643, Z -3.0000, A 0.000, B 0.000, C 0.000 }
gfCNCPoint2[9943] = {X 302.8089, Y 48.4400, Z -3.0000, A 0.000, B 0.000, C 0.000 }
gfCNCPoint2[9944] = {X 302.1122, Y 47.7433, Z -3.0000, A 0.000, B 0.000, C 0.000 }
gfCNCPoint2[9945] = {X 301.5880, Y 46.9091, Z -3.0000, A 0.000, B 0.000, C 0.000 }
gfCNCPoint2[9946] = {X 301.2626, Y 45.9791, Z -3.0000, A 0.000, B 0.000, C 0.000 }
gfCNCPoint2[9947] = {X 301.1523, Y 45.0000, Z -3.0000, A 0.000, B 0.000, C 0.000 }
gfCNCPoint2[9948] = {X 301.1524, Y 44.1992, Z -3.0000, A 0.000, B 0.000, C 0.000 }
gfCNCPoint2[9949] = {X 301.2703, Y 43.2558, Z -3.0000, A 0.000, B 0.000, C 0.000 }
gfCNCPoint2[9950] = {X 301.5735, Y 42.3546, Z -3.0000, A 0.000, B 0.000, C 0.000 }
gfCNCPoint2[9951] = {X 302.0499, Y 41.5318, Z -3.0000, A 0.000, B 0.000, C 0.000 }
gfCNCPoint2[9952] = {X 302.6804, Y 40.8202, Z -3.0000, A 0.000, B 0.000, C 0.000 }
gfCNCPoint2[9953] = {X 302.6804, Y 34.1143, Z -3.0000, A 0.000, B 0.000, C 0.000 }
gfCNCPoint2[9954] = {X 293.9340, Y 34.1143, Z -3.0000, A 0.000, B 0.000, C 0.000 }
gfCNCPoint2[9955] = {X 293.9331, Y 40.8663, Z -3.0000, A 0.000, B 0.000, C 0.000 }
gfCNCPoint2[9956] = {X 294.5730, Y 41.5612, Z -3.0000, A 0.000, B 0.000, C 0.000 }
gfCNCPoint2[9957] = {X 295.0538, Y 42.3745, Z -3.0000, A 0.000, B 0.000, C 0.000 }
gfCNCPoint2[9958] = {X 295.3543, Y 43.2702, Z -3.0000, A 0.000, B 0.000, C 0.000 }
gfCNCPoint2[9959] = {X 295.4611, Y 44.2089, Z -3.0000, A 0.000, B 0.000, C 0.000 }
gfCNCPoint2[9960] = {X 295.4611, Y 45.0000, Z -3.0000, A 0.000, B 0.000, C 0.000 }
gfCNCPoint2[9961] = {X 295.3508, Y 45.9791, Z -3.0000, A 0.000, B 0.000, C 0.000 }
gfCNCPoint2[9962] = {X 295.0254, Y 46.9091, Z -3.0000, A 0.000, B 0.000, C 0.000 }
gfCNCPoint2[9963] = {X 294.5012, Y 47.7434, Z -3.0000, A 0.000, B 0.000, C 0.000 }
gfCNCPoint2[9964] = {X 293.8045, Y 48.4401, Z -3.0000, A 0.000, B 0.000, C 0.000 }
gfCNCPoint2[9965] = {X 292.9702, Y 48.9643, Z -3.0000, A 0.000, B 0.000, C 0.000 }
gfCNCPoint2[9966] = {X 292.0402, Y 49.2897, Z -3.0000, A 0.000, B 0.000, C 0.000 }
gfCNCPoint2[9967] = {X 291.0611, Y 49.4000, Z -3.0000, A 0.000, B 0.000, C 0.000 }
gfCNCPoint2[9968] = {X 284.6177, Y 49.4000, Z -3.0000, A 0.000, B 0.000, C 0.000 }
gfCNCPoint2[9969] = {X 283.6386, Y 49.2897, Z -3.0000, A 0.000, B 0.000, C 0.000 }
gfCNCPoint2[9970] = {X 282.7086, Y 48.9643, Z -3.0000, A 0.000, B 0.000, C 0.000 }
gfCNCPoint2[9971] = {X 281.8743, Y 48.4400, Z -3.0000, A 0.000, B 0.000, C 0.000 }
gfCNCPoint2[9972] = {X 281.1776, Y 47.7433, Z -3.0000, A 0.000, B 0.000, C 0.000 }
gfCNCPoint2[9973] = {X 280.6534, Y 46.9091, Z -3.0000, A 0.000, B 0.000, C 0.000 }
gfCNCPoint2[9974] = {X 280.3280, Y 45.9791, Z -3.0000, A 0.000, B 0.000, C 0.000 }
gfCNCPoint2[9975] = {X 280.2177, Y 45.0000, Z -3.0000, A 0.000, B 0.000, C 0.000 }
gfCNCPoint2[9976] = {X 280.2177, Y 44.2066, Z -3.0000, A 0.000, B 0.000, C 0.000 }
gfCNCPoint2[9977] = {X 280.3228, Y 43.2697, Z -3.0000, A 0.000, B 0.000, C 0.000 }
gfCNCPoint2[9978] = {X 280.6229, Y 42.3760, Z -3.0000, A 0.000, B 0.000, C 0.000 }
gfCNCPoint2[9979] = {X 281.1045, Y 41.5655, Z -3.0000, A 0.000, B 0.000, C 0.000 }
gfCNCPoint2[9980] = {X 281.7459, Y 40.8746, Z -3.0000, A 0.000, B 0.000, C 0.000 }
gfCNCPoint2[9981] = {X 281.7455, Y 16.3113, Z -3.0000, A 0.000, B 0.000, C 0.000 }
gfCNCPoint2[9982] = {X 281.1008, Y 15.6221, Z -3.0000, A 0.000, B 0.000, C 0.000 }
gfCNCPoint2[9983] = {X 280.6178, Y 14.8114, Z -3.0000, A 0.000, B 0.000, C 0.000 }
gfCNCPoint2[9984] = {X 280.3189, Y 13.9162, Z -3.0000, A 0.000, B 0.000, C 0.000 }
gfCNCPoint2[9985] = {X 280.2177, Y 12.9779, Z -3.0000, A 0.000, B 0.000, C 0.000 }
gfCNCPoint2[9986] = {X 280.2177, Y 12.1868, Z -3.0000, A 0.000, B 0.000, C 0.000 }
gfCNCPoint2[9987] = {X 280.3280, Y 11.2077, Z -3.0000, A 0.000, B 0.000, C 0.000 }
gfCNCPoint2[9988] = {X 280.6534, Y 10.2777, Z -3.0000, A 0.000, B 0.000, C 0.000 }
gfCNCPoint2[9989] = {X 281.1776, Y 9.4435, Z -3.0000, A 0.000, B 0.000, C 0.000 }
gfCNCPoint2[9990] = {X 281.8743, Y 8.7468, Z -3.0000, A 0.000, B 0.000, C 0.000 }
gfCNCPoint2[9991] = {X 282.7086, Y 8.2226, Z -3.0000, A 0.000, B 0.000, C 0.000 }
gfCNCPoint2[9992] = {X 283.6386, Y 7.8971, Z -3.0000, A 0.000, B 0.000, C 0.000 }
gfCNCPoint2[9993] = {X 284.6177, Y 7.7868, Z -3.0000, A 0.000, B 0.000, C 0.000 }
gfCNCPoint2[9994] = {X 291.0611, Y 7.7868, Z -3.0000, A 0.000, B 0.000, C 0.000 }
gfCNCPoint2[9995] = {X 292.0402, Y 7.8971, Z -3.0000, A 0.000, B 0.000, C 0.000 }
gfCNCPoint2[9996] = {X 292.9702, Y 8.2226, Z -3.0000, A 0.000, B 0.000, C 0.000 }
gfCNCPoint2[9997] = {X 293.8045, Y 8.7468, Z -3.0000, A 0.000, B 0.000, C 0.000 }
gfCNCPoint2[9998] = {X 294.5012, Y 9.4435, Z -3.0000, A 0.000, B 0.000, C 0.000 }
gfCNCPoint2[9999] = {X 295.0254, Y 10.2777, Z -3.0000, A 0.000, B 0.000, C 0.000 }
gfCNCPoint2[10000] = {X 295.3508, Y 11.2077, Z -3.0000, A 0.000, B 0.000, C 0.000 }
gfCNCPoint2[10001] = {X 295.4611, Y 12.1868, Z -3.0000, A 0.000, B 0.000, C 0.000 }
gfCNCPoint2[10002] = {X 295.4609, Y 13.0233, Z -3.0000, A 0.000, B 0.000, C 0.000 }
gfCNCPoint2[10003] = {X 295.3525, Y 13.9495, Z -3.0000, A 0.000, B 0.000, C 0.000 }
gfCNCPoint2[10004] = {X 295.0514, Y 14.8321, Z -3.0000, A 0.000, B 0.000, C 0.000 }
gfCNCPoint2[10005] = {X 294.5710, Y 15.6314, Z -3.0000, A 0.000, B 0.000, C 0.000 }
gfCNCPoint2[10006] = {X 293.9330, Y 16.3116, Z -3.0000, A 0.000, B 0.000, C 0.000 }
gfCNCPoint2[10007] = {X 293.9342, Y 22.1165, Z -3.0000, A 0.000, B 0.000, C 0.000 }
gfCNCPoint2[10008] = {X 302.6795, Y 22.1165, Z -3.0000, A 0.000, B 0.000, C 0.000 }
gfCNCPoint2[10009] = {X 302.6800, Y 16.3112, Z -3.0000, A 0.000, B 0.000, C 0.000 }
gfCNCPoint2[10010] = {X 302.0353, Y 15.6221, Z -3.0000, A 0.000, B 0.000, C 0.000 }
gfCNCPoint2[10011] = {X 301.5524, Y 14.8113, Z -3.0000, A 0.000, B 0.000, C 0.000 }
gfCNCPoint2[10012] = {X 301.2534, Y 13.9162, Z -3.0000, A 0.000, B 0.000, C 0.000 }
gfCNCPoint2[10013] = {X 301.1523, Y 12.9779, Z -3.0000, A 0.000, B 0.000, C 0.000 }
gfCNCPoint2[10014] = {X 301.1523, Y 12.1868, Z -3.0000, A 0.000, B 0.000, C 0.000 }
gfCNCPoint2[10015] = {X 301.2626, Y 11.2077, Z -3.0000, A 0.000, B 0.000, C 0.000 }
gfCNCPoint2[10016] = {X 301.5880, Y 10.2777, Z -3.0000, A 0.000, B 0.000, C 0.000 }
gfCNCPoint2[10017] = {X 302.1122, Y 9.4435, Z -3.0000, A 0.000, B 0.000, C 0.000 }
gfCNCPoint2[10018] = {X 302.8089, Y 8.7468, Z -3.0000, A 0.000, B 0.000, C 0.000 }
gfCNCPoint2[10019] = {X 303.6432, Y 8.2226, Z -3.0000, A 0.000, B 0.000, C 0.000 }
gfCNCPoint2[10020] = {X 304.5732, Y 7.8971, Z -3.0000, A 0.000, B 0.000, C 0.000 }
gfCNCPoint2[10021] = {X 305.5523, Y 7.7868, Z -3.0000, A 0.000, B 0.000, C 0.000 }
gfCNCPoint2[10022] = {X 311.9957, Y 7.7868, Z -3.0000, A 0.000, B 0.000, C 0.000 }
gfCNCPoint2[10023] = {X 312.9748, Y 7.8971, Z -3.0000, A 0.000, B 0.000, C 0.000 }
gfCNCPoint2[10024] = {X 313.9048, Y 8.2226, Z -3.0000, A 0.000, B 0.000, C 0.000 }
gfCNCPoint2[10025] = {X 314.7391, Y 8.7468, Z -3.0000, A 0.000, B 0.000, C 0.000 }
gfCNCPoint2[10026] = {X 315.4358, Y 9.4435, Z -3.0000, A 0.000, B 0.000, C 0.000 }
gfCNCPoint2[10027] = {X 315.9600, Y 10.2777, Z -3.0000, A 0.000, B 0.000, C 0.000 }
gfCNCPoint2[10028] = {X 316.2854, Y 11.2077, Z -3.0000, A 0.000, B 0.000, C 0.000 }
gfCNCPoint2[10029] = {X 316.3957, Y 12.1868, Z -3.0000, A 0.000, B 0.000, C 0.000 }
gfCNCPoint2[10030] = {X 316.3955, Y 13.0233, Z -3.0000, A 0.000, B 0.000, C 0.000 }
gfCNCPoint2[10031] = {X 316.2871, Y 13.9495, Z -3.0000, A 0.000, B 0.000, C 0.000 }
gfCNCPoint2[10032] = {X 315.9860, Y 14.8320, Z -3.0000, A 0.000, B 0.000, C 0.000 }
gfCNCPoint2[10033] = {X 315.5057, Y 15.6313, Z -3.0000, A 0.000, B 0.000, C 0.000 }
gfCNCPoint2[10034] = {X 314.8677, Y 16.3114, Z -3.0000, A 0.000, B 0.000, C 0.000 }
gfCNCPoint2[10035] = {X 314.8675, Y 40.8752, Z -3.0000, A 0.000, B 0.000, C 0.000 }
gfCNCPoint2[10036] = {X 315.5124, Y 41.5644, Z -3.0000, A 0.000, B 0.000, C 0.000 }
gfCNCPoint2[10037] = {X 315.9955, Y 42.3752, Z -3.0000, A 0.000, B 0.000, C 0.000 }
gfCNCPoint2[10038] = {X 316.2945, Y 43.2705, Z -3.0000, A 0.000, B 0.000, C 0.000 }
gfCNCPoint2[10039] = {X 316.3957, Y 44.2089, Z -3.0000, A 0.000, B 0.000, C 0.000 }
gfCNCPoint2[10040] = {X 316.3957, Y 45.0000, Z -3.0000, A 0.000, B 0.000, C 0.000 }
gfCNCPoint2[10041] = {X 316.3190, Y 45.8182, Z -3.0000, A 0.000, B 0.000, C 0.000 }
gfCNCPoint2[10042] = {X 316.0914, Y 46.6079, Z -3.0000, A 0.000, B 0.000, C 0.000 }
gfCNCPoint2[10043] = {X 315.7209, Y 47.3415, Z -3.0000, A 0.000, B 0.000, C 0.000 }
gfCNCPoint2[10044] = {X 315.2205, Y 47.9934, Z -3.0000, A 0.000, B 0.000, C 0.000 }
gfCNCPoint2[10045] = {X 315.5723, Y 48.3200, Z -3.0000, A 0.000, B 0.000, C 0.000 }
gfCNCPoint2[10046] = {X 324.3107, Y 48.3200, Z -3.0000, A 0.000, B 0.000, C 0.000 }
gfCNCPoint2[10047] = {X 325.5555, Y 48.4004, Z -3.0000, A 0.000, B 0.000, C 0.000 }
gfCNCPoint2[10048] = {X 326.7797, Y 48.6402, Z -3.0000, A 0.000, B 0.000, C 0.000 }
gfCNCPoint2[10049] = {X 325.5882, Y 48.0963, Z -3.0000, A 0.000, B 0.000, C 0.000 }
gfCNCPoint2[10050] = {X 324.4810, Y 47.3966, Z -3.0000, A 0.000, B 0.000, C 0.000 }
gfCNCPoint2[10051] = {X 323.4784, Y 46.5538, Z -3.0000, A 0.000, B 0.000, C 0.000 }
gfCNCPoint2[10052] = {X 322.8382, Y 45.9295, Z -3.0000, A 0.000, B 0.000, C 0.000 }
gfCNCPoint2[10053] = {X 322.2180, Y 45.2650, Z -3.0000, A 0.000, B 0.000, C 0.000 }
gfCNCPoint2[10054] = {X 321.6628, Y 44.5452, Z -3.0000, A 0.000, B 0.000, C 0.000 }
gfCNCPoint2[10055] = {X 323.6300, Y 43.1703, Z -3.0000, A 0.000, B 0.000, C 0.000 }
gfCNCPoint2[10056] = {X 323.0063, Y 42.0918, Z -3.0000, A 0.000, B 0.000, C 0.000 }
gfCNCPoint2[10057] = {X 322.5757, Y 40.9227, Z -3.0000, A 0.000, B 0.000, C 0.000 }
gfCNCPoint2[10058] = {X 322.3506, Y 39.6973, Z -3.0000, A 0.000, B 0.000, C 0.000 }
gfCNCPoint2[10059] = {X 322.3379, Y 38.4514, Z -3.0000, A 0.000, B 0.000, C 0.000 }
gfCNCPoint2[10060] = {X 322.5377, Y 37.2217, Z -3.0000, A 0.000, B 0.000, C 0.000 }
gfCNCPoint2[10061] = {X 322.9443, Y 36.0440, Z -3.0000, A 0.000, B 0.000, C 0.000 }
gfCNCPoint2[10062] = {X 323.5458, Y 34.9529, Z -3.0000, A 0.000, B 0.000, C 0.000 }
gfCNCPoint2[10063] = {X 327.7790, Y 28.6234, Z -3.0000, A 0.000, B 0.000, C 0.000 }
gfCNCPoint2[10064] = {X 328.5158, Y 27.6951, Z -3.0000, A 0.000, B 0.000, C 0.000 }
gfCNCPoint2[10065] = {X 329.3936, Y 26.8986, Z -3.0000, A 0.000, B 0.000, C 0.000 }
gfCNCPoint2[10066] = {X 330.3889, Y 26.2552, Z -3.0000, A 0.000, B 0.000, C 0.000 }
gfCNCPoint2[10067] = {X 331.5063, Y 25.7713, Z -3.0000, A 0.000, B 0.000, C 0.000 }
gfCNCPoint2[10068] = {X 332.6887, Y 25.4804, Z -3.0000, A 0.000, B 0.000, C 0.000 }
gfCNCPoint2[10069] = {X 333.9031, Y 25.3907, Z -3.0000, A 0.000, B 0.000, C 0.000 }
gfCNCPoint2[10070] = {X 335.1154, Y 25.5046, Z -3.0000, A 0.000, B 0.000, C 0.000 }
gfCNCPoint2[10071] = {X 336.2918, Y 25.8191, Z -3.0000, A 0.000, B 0.000, C 0.000 }
gfCNCPoint2[10072] = {X 337.3993, Y 26.3252, Z -3.0000, A 0.000, B 0.000, C 0.000 }
gfCNCPoint2[10073] = {X 338.1754, Y 26.8291, Z -3.0000, A 0.000, B 0.000, C 0.000 }
gfCNCPoint2[10074] = {X 338.8813, Y 27.4275, Z -3.0000, A 0.000, B 0.000, C 0.000 }
gfCNCPoint2[10075] = {X 339.4514, Y 27.9767, Z -3.0000, A 0.000, B 0.000, C 0.000 }
gfCNCPoint2[10076] = {X 339.8232, Y 28.3622, Z -3.0000, A 0.000, B 0.000, C 0.000 }
gfCNCPoint2[10077] = {X 340.1656, Y 28.7740, Z -3.0000, A 0.000, B 0.000, C 0.000 }
gfCNCPoint2[10078] = {X 345.8671, Y 24.3770, Z -3.0000, A 0.000, B 0.000, C 0.000 }
gfCNCPoint2[10079] = {X 346.4661, Y 25.2135, Z -3.0000, A 0.000, B 0.000, C 0.000 }
gfCNCPoint2[10080] = {X 347.0041, Y 26.0905, Z -3.0000, A 0.000, B 0.000, C 0.000 }
gfCNCPoint2[10081] = {X 347.1181, Y 24.7344, Z -3.0000, A 0.000, B 0.000, C 0.000 }
gfCNCPoint2[10082] = {X 346.9942, Y 23.3793, Z -3.0000, A 0.000, B 0.000, C 0.000 }
gfCNCPoint2[10083] = {X 346.9501, Y 23.1695, Z -3.0000, A 0.000, B 0.000, C 0.000 }
gfCNCPoint2[10084] = {X 346.8820, Y 22.9664, Z -3.0000, A 0.000, B 0.000, C 0.000 }
gfCNCPoint2[10085] = {X 346.3957, Y 23.6869, Z -3.0000, A 0.000, B 0.000, C 0.000 }
gfCNCPoint2[10086] = {X 345.8671, Y 24.3770, Z -3.0000, A 0.000, B 0.000, C 0.000 }
gfCNCPoint2[10087] = {X 343.9666, Y 25.8427, Z -3.0000, A 0.000, B 0.000, C 0.000 }
gfCNCPoint2[10088] = {X 344.4663, Y 26.5405, Z -3.0000, A 0.000, B 0.000, C 0.000 }
gfCNCPoint2[10089] = {X 344.9152, Y 27.2721, Z -3.0000, A 0.000, B 0.000, C 0.000 }
gfCNCPoint2[10090] = {X 345.4669, Y 28.3755, Z -3.0000, A 0.000, B 0.000, C 0.000 }
gfCNCPoint2[10091] = {X 345.9033, Y 29.5293, Z -3.0000, A 0.000, B 0.000, C 0.000 }
gfCNCPoint2[10092] = {X 346.4600, Y 29.6320, Z -3.0000, A 0.000, B 0.000, C 0.000 }
gfCNCPoint2[10093] = {X 347.0261, Y 29.6228, Z -3.0000, A 0.000, B 0.000, C 0.000 }
gfCNCPoint2[10094] = {X 347.4357, Y 29.5576, Z -3.0000, A 0.000, B 0.000, C 0.000 }
gfCNCPoint2[10095] = {X 347.7945, Y 29.3497, Z -3.0000, A 0.000, B 0.000, C 0.000 }
gfCNCPoint2[10096] = {X 348.4751, Y 28.6299, Z -3.0000, A 0.000, B 0.000, C 0.000 }
gfCNCPoint2[10097] = {X 348.9860, Y 27.7811, Z -3.0000, A 0.000, B 0.000, C 0.000 }
gfCNCPoint2[10098] = {X 349.3035, Y 26.8428, Z -3.0000, A 0.000, B 0.000, C 0.000 }
gfCNCPoint2[10099] = {X 349.3377, Y 26.6716, Z -3.0000, A 0.000, B 0.000, C 0.000 }
gfCNCPoint2[10100] = {X 349.3689, Y 26.4998, Z -3.0000, A 0.000, B 0.000, C 0.000 }
gfCNCPoint2[10101] = {X 349.5024, Y 25.3283, Z -3.0000, A 0.000, B 0.000, C 0.000 }
gfCNCPoint2[10102] = {X 349.4996, Y 24.1493, Z -3.0000, A 0.000, B 0.000, C 0.000 }
gfCNCPoint2[10103] = {X 349.3605, Y 22.9785, Z -3.0000, A 0.000, B 0.000, C 0.000 }
gfCNCPoint2[10104] = {X 349.1887, Y 22.2867, Z -3.0000, A 0.000, B 0.000, C 0.000 }
gfCNCPoint2[10105] = {X 348.9033, Y 21.6336, Z -3.0000, A 0.000, B 0.000, C 0.000 }
gfCNCPoint2[10106] = {X 348.5126, Y 21.0375, Z -3.0000, A 0.000, B 0.000, C 0.000 }
gfCNCPoint2[10107] = {X 348.1201, Y 20.6782, Z -3.0000, A 0.000, B 0.000, C 0.000 }
gfCNCPoint2[10108] = {X 347.6259, Y 20.4810, Z -3.0000, A 0.000, B 0.000, C 0.000 }
gfCNCPoint2[10109] = {X 346.5728, Y 20.3825, Z -3.0000, A 0.000, B 0.000, C 0.000 }
gfCNCPoint2[10110] = {X 345.5200, Y 20.4828, Z -3.0000, A 0.000, B 0.000, C 0.000 }
gfCNCPoint2[10111] = {X 344.7178, Y 21.8936, Z -3.0000, A 0.000, B 0.000, C 0.000 }
gfCNCPoint2[10112] = {X 343.7338, Y 23.1841, Z -3.0000, A 0.000, B 0.000, C 0.000 }
gfCNCPoint2[10113] = {X 342.5857, Y 24.3311, Z -3.0000, A 0.000, B 0.000, C 0.000 }
gfCNCPoint2[10114] = {X 342.7815, Y 24.5198, Z -3.0000, A 0.000, B 0.000, C 0.000 }
gfCNCPoint2[10115] = {X 343.3984, Y 25.1594, Z -3.0000, A 0.000, B 0.000, C 0.000 }
gfCNCPoint2[10116] = {X 343.9666, Y 25.8427, Z -3.0000, A 0.000, B 0.000, C 0.000 }
gfCNCPoint2[10117] = {X 342.0661, Y 27.3083, Z -3.0000, A 0.000, B 0.000, C 0.000 }
gfCNCPoint2[10118] = {X 342.8614, Y 28.5165, Z -3.0000, A 0.000, B 0.000, C 0.000 }
gfCNCPoint2[10119] = {X 343.4678, Y 29.8297, Z -3.0000, A 0.000, B 0.000, C 0.000 }
gfCNCPoint2[10120] = {X 343.8717, Y 31.2186, Z -3.0000, A 0.000, B 0.000, C 0.000 }
gfCNCPoint2[10121] = {X 344.6368, Y 31.6215, Z -3.0000, A 0.000, B 0.000, C 0.000 }
gfCNCPoint2[10122] = {X 345.4576, Y 31.8935, Z -3.0000, A 0.000, B 0.000, C 0.000 }
gfCNCPoint2[10123] = {X 346.3120, Y 32.0272, Z -3.0000, A 0.000, B 0.000, C 0.000 }
gfCNCPoint2[10124] = {X 347.1766, Y 32.0191, Z -3.0000, A 0.000, B 0.000, C 0.000 }
gfCNCPoint2[10125] = {X 347.9589, Y 31.9043, Z -3.0000, A 0.000, B 0.000, C 0.000 }
gfCNCPoint2[10126] = {X 348.6961, Y 31.6186, Z -3.0000, A 0.000, B 0.000, C 0.000 }
gfCNCPoint2[10127] = {X 349.3513, Y 31.1762, Z -3.0000, A 0.000, B 0.000, C 0.000 }
gfCNCPoint2[10128] = {X 350.1528, Y 30.3725, Z -3.0000, A 0.000, B 0.000, C 0.000 }
gfCNCPoint2[10129] = {X 350.8140, Y 29.4498, Z -3.0000, A 0.000, B 0.000, C 0.000 }
gfCNCPoint2[10130] = {X 351.3174, Y 28.4325, Z -3.0000, A 0.000, B 0.000, C 0.000 }
gfCNCPoint2[10131] = {X 351.6499, Y 27.3472, Z -3.0000, A 0.000, B 0.000, C 0.000 }
gfCNCPoint2[10132] = {X 351.8783, Y 25.7641, Z -3.0000, A 0.000, B 0.000, C 0.000 }
gfCNCPoint2[10133] = {X 351.9039, Y 24.1649, Z -3.0000, A 0.000, B 0.000, C 0.000 }
gfCNCPoint2[10134] = {X 351.7265, Y 22.5753, Z -3.0000, A 0.000, B 0.000, C 0.000 }
gfCNCPoint2[10135] = {X 351.4576, Y 21.5045, Z -3.0000, A 0.000, B 0.000, C 0.000 }
gfCNCPoint2[10136] = {X 351.0150, Y 20.4930, Z -3.0000, A 0.000, B 0.000, C 0.000 }
gfCNCPoint2[10137] = {X 350.4108, Y 19.5689, Z -3.0000, A 0.000, B 0.000, C 0.000 }
gfCNCPoint2[10138] = {X 349.7598, Y 18.9041, Z -3.0000, A 0.000, B 0.000, C 0.000 }
gfCNCPoint2[10139] = {X 348.9693, Y 18.4135, Z -3.0000, A 0.000, B 0.000, C 0.000 }
gfCNCPoint2[10140] = {X 348.0846, Y 18.1252, Z -3.0000, A 0.000, B 0.000, C 0.000 }
gfCNCPoint2[10141] = {X 346.9931, Y 17.9932, Z -3.0000, A 0.000, B 0.000, C 0.000 }
gfCNCPoint2[10142] = {X 345.8938, Y 18.0116, Z -3.0000, A 0.000, B 0.000, C 0.000 }
gfCNCPoint2[10143] = {X 344.8074, Y 18.1802, Z -3.0000, A 0.000, B 0.000, C 0.000 }
gfCNCPoint2[10144] = {X 343.7542, Y 18.4957, Z -3.0000, A 0.000, B 0.000, C 0.000 }
gfCNCPoint2[10145] = {X 343.2661, Y 19.6260, Z -3.0000, A 0.000, B 0.000, C 0.000 }
gfCNCPoint2[10146] = {X 342.6385, Y 20.6851, Z -3.0000, A 0.000, B 0.000, C 0.000 }
gfCNCPoint2[10147] = {X 341.8815, Y 21.6561, Z -3.0000, A 0.000, B 0.000, C 0.000 }
gfCNCPoint2[10148] = {X 341.0073, Y 22.5231, Z -3.0000, A 0.000, B 0.000, C 0.000 }
gfCNCPoint2[10149] = {X 340.7217, Y 22.7629, Z -3.0000, A 0.000, B 0.000, C 0.000 }
gfCNCPoint2[10150] = {X 340.4270, Y 22.9916, Z -3.0000, A 0.000, B 0.000, C 0.000 }
gfCNCPoint2[10151] = {X 339.6615, Y 23.5549, Z -3.0000, A 0.000, B 0.000, C 0.000 }
gfCNCPoint2[10152] = {X 339.1299, Y 23.9121, Z -3.0000, A 0.000, B 0.000, C 0.000 }
gfCNCPoint2[10153] = {X 338.5759, Y 24.2333, Z -3.0000, A 0.000, B 0.000, C 0.000 }
gfCNCPoint2[10154] = {X 339.6078, Y 24.9035, Z -3.0000, A 0.000, B 0.000, C 0.000 }
gfCNCPoint2[10155] = {X 340.5464, Y 25.6991, Z -3.0000, A 0.000, B 0.000, C 0.000 }
gfCNCPoint2[10156] = {X 341.1164, Y 26.2482, Z -3.0000, A 0.000, B 0.000, C 0.000 }
gfCNCPoint2[10157] = {X 341.6108, Y 26.7608, Z -3.0000, A 0.000, B 0.000, C 0.000 }
gfCNCPoint2[10158] = {X 342.0661, Y 27.3083, Z -3.0000, A 0.000, B 0.000, C 0.000 }
gfCNCPoint2[10159] = {X 340.1656, Y 28.7740, Z -3.0000, A 0.000, B 0.000, C 0.000 }
gfCNCPoint2[10160] = {X 340.7341, Y 29.6298, Z -3.0000, A 0.000, B 0.000, C 0.000 }
gfCNCPoint2[10161] = {X 341.1764, Y 30.5572, Z -3.0000, A 0.000, B 0.000, C 0.000 }
gfCNCPoint2[10162] = {X 341.4838, Y 31.5376, Z -3.0000, A 0.000, B 0.000, C 0.000 }
gfCNCPoint2[10163] = {X 341.6501, Y 32.5514, Z -3.0000, A 0.000, B 0.000, C 0.000 }
gfCNCPoint2[10164] = {X 341.8444, Y 32.7092, Z -3.0000, A 0.000, B 0.000, C 0.000 }
gfCNCPoint2[10165] = {X 342.0409, Y 32.8642, Z -3.0000, A 0.000, B 0.000, C 0.000 }
gfCNCPoint2[10166] = {X 342.9838, Y 33.4816, Z -3.0000, A 0.000, B 0.000, C 0.000 }
gfCNCPoint2[10167] = {X 344.0071, Y 33.9538, Z -3.0000, A 0.000, B 0.000, C 0.000 }
gfCNCPoint2[10168] = {X 345.0887, Y 34.2707, Z -3.0000, A 0.000, B 0.000, C 0.000 }
gfCNCPoint2[10169] = {X 346.2050, Y 34.4254, Z -3.0000, A 0.000, B 0.000, C 0.000 }
gfCNCPoint2[10170] = {X 347.3320, Y 34.4145, Z -3.0000, A 0.000, B 0.000, C 0.000 }
gfCNCPoint2[10171] = {X 348.3016, Y 34.2891, Z -3.0000, A 0.000, B 0.000, C 0.000 }
gfCNCPoint2[10172] = {X 349.2374, Y 34.0062, Z -3.0000, A 0.000, B 0.000, C 0.000 }
gfCNCPoint2[10173] = {X 350.1141, Y 33.5736, Z -3.0000, A 0.000, B 0.000, C 0.000 }
gfCNCPoint2[10174] = {X 350.9079, Y 33.0030, Z -3.0000, A 0.000, B 0.000, C 0.000 }
gfCNCPoint2[10175] = {X 351.7846, Y 32.1517, Z -3.0000, A 0.000, B 0.000, C 0.000 }
gfCNCPoint2[10176] = {X 352.5435, Y 31.1939, Z -3.0000, A 0.000, B 0.000, C 0.000 }
gfCNCPoint2[10177] = {X 353.1718, Y 30.1458, Z -3.0000, A 0.000, B 0.000, C 0.000 }
gfCNCPoint2[10178] = {X 353.6589, Y 29.0251, Z -3.0000, A 0.000, B 0.000, C 0.000 }
gfCNCPoint2[10179] = {X 353.9965, Y 27.8507, Z -3.0000, A 0.000, B 0.000, C 0.000 }
gfCNCPoint2[10180] = {X 354.2239, Y 26.4407, Z -3.0000, A 0.000, B 0.000, C 0.000 }
gfCNCPoint2[10181] = {X 354.3160, Y 25.0155, Z -3.0000, A 0.000, B 0.000, C 0.000 }
gfCNCPoint2[10182] = {X 354.2720, Y 23.5880, Z -3.0000, A 0.000, B 0.000, C 0.000 }
gfCNCPoint2[10183] = {X 354.0923, Y 22.1712, Z -3.0000, A 0.000, B 0.000, C 0.000 }
gfCNCPoint2[10184] = {X 353.8396, Y 21.0759, Z -3.0000, A 0.000, B 0.000, C 0.000 }
gfCNCPoint2[10185] = {X 353.4529, Y 20.0203, Z -3.0000, A 0.000, B 0.000, C 0.000 }
gfCNCPoint2[10186] = {X 352.9383, Y 19.0210, Z -3.0000, A 0.000, B 0.000, C 0.000 }
gfCNCPoint2[10187] = {X 352.3035, Y 18.0932, Z -3.0000, A 0.000, B 0.000, C 0.000 }
gfCNCPoint2[10188] = {X 351.5366, Y 17.2659, Z -3.0000, A 0.000, B 0.000, C 0.000 }
gfCNCPoint2[10189] = {X 350.6340, Y 16.5891, Z -3.0000, A 0.000, B 0.000, C 0.000 }
gfCNCPoint2[10190] = {X 349.6249, Y 16.0848, Z -3.0000, A 0.000, B 0.000, C 0.000 }
gfCNCPoint2[10191] = {X 348.5419, Y 15.7692, Z -3.0000, A 0.000, B 0.000, C 0.000 }
gfCNCPoint2[10192] = {X 347.1562, Y 15.5985, Z -3.0000, A 0.000, B 0.000, C 0.000 }
gfCNCPoint2[10193] = {X 345.7601, Y 15.6146, Z -3.0000, A 0.000, B 0.000, C 0.000 }
gfCNCPoint2[10194] = {X 344.3786, Y 15.8171, Z -3.0000, A 0.000, B 0.000, C 0.000 }
gfCNCPoint2[10195] = {X 343.0367, Y 16.2024, Z -3.0000, A 0.000, B 0.000, C 0.000 }
gfCNCPoint2[10196] = {X 341.7582, Y 16.7636, Z -3.0000, A 0.000, B 0.000, C 0.000 }
gfCNCPoint2[10197] = {X 341.3708, Y 18.0082, Z -3.0000, A 0.000, B 0.000, C 0.000 }
gfCNCPoint2[10198] = {X 340.7676, Y 19.1638, Z -3.0000, A 0.000, B 0.000, C 0.000 }
gfCNCPoint2[10199] = {X 339.9680, Y 20.1932, Z -3.0000, A 0.000, B 0.000, C 0.000 }
gfCNCPoint2[10200] = {X 338.9976, Y 21.0636, Z -3.0000, A 0.000, B 0.000, C 0.000 }
gfCNCPoint2[10201] = {X 338.2497, Y 21.6140, Z -3.0000, A 0.000, B 0.000, C 0.000 }
gfCNCPoint2[10202] = {X 337.8538, Y 21.8795, Z -3.0000, A 0.000, B 0.000, C 0.000 }
gfCNCPoint2[10203] = {X 337.4413, Y 22.1185, Z -3.0000, A 0.000, B 0.000, C 0.000 }
gfCNCPoint2[10204] = {X 336.3239, Y 22.6023, Z -3.0000, A 0.000, B 0.000, C 0.000 }
gfCNCPoint2[10205] = {X 335.1415, Y 22.8932, Z -3.0000, A 0.000, B 0.000, C 0.000 }
gfCNCPoint2[10206] = {X 333.9271, Y 22.9829, Z -3.0000, A 0.000, B 0.000, C 0.000 }
gfCNCPoint2[10207] = {X 332.7148, Y 22.8690, Z -3.0000, A 0.000, B 0.000, C 0.000 }
gfCNCPoint2[10208] = {X 331.5384, Y 22.5546, Z -3.0000, A 0.000, B 0.000, C 0.000 }
gfCNCPoint2[10209] = {X 330.4309, Y 22.0485, Z -3.0000, A 0.000, B 0.000, C 0.000 }
gfCNCPoint2[10210] = {X 329.5143, Y 21.4374, Z -3.0000, A 0.000, B 0.000, C 0.000 }
gfCNCPoint2[10211] = {X 328.7005, Y 20.6949, Z -3.0000, A 0.000, B 0.000, C 0.000 }
gfCNCPoint2[10212] = {X 328.0080, Y 19.8382, Z -3.0000, A 0.000, B 0.000, C 0.000 }
gfCNCPoint2[10213] = {X 327.4528, Y 18.8869, Z -3.0000, A 0.000, B 0.000, C 0.000 }
gfCNCPoint2[10214] = {X 323.9321, Y 11.6443, Z -3.0000, A 0.000, B 0.000, C 0.000 }
gfCNCPoint2[10215] = {X 323.5337, Y 10.6422, Z -3.0000, A 0.000, B 0.000, C 0.000 }
gfCNCPoint2[10216] = {X 323.2878, Y 9.5922, Z -3.0000, A 0.000, B 0.000, C 0.000 }
gfCNCPoint2[10217] = {X 323.1997, Y 8.5174, Z -3.0000, A 0.000, B 0.000, C 0.000 }
gfCNCPoint2[10218] = {X 323.2713, Y 7.4414, Z -3.0000, A 0.000, B 0.000, C 0.000 }
gfCNCPoint2[10219] = {X 323.4719, Y 6.4885, Z -3.0000, A 0.000, B 0.000, C 0.000 }
gfCNCPoint2[10220] = {X 323.7980, Y 5.5709, Z -3.0000, A 0.000, B 0.000, C 0.000 }
gfCNCPoint2[10221] = {X 324.2435, Y 4.7050, Z -3.0000, A 0.000, B 0.000, C 0.000 }
gfCNCPoint2[10222] = {X 168.0205, Y 4.7050, Z -3.0000, A 0.000, B 0.000, C 0.000 }
gfCNCPoint2[10223] = {X 168.0205, Y 9.5050, Z -3.0000, A 0.000, B 0.000, C 0.000 }
gfCNCPoint2[10224] = {X 166.5360, Y 9.5050, Z -3.0000, A 0.000, B 0.000, C 0.000 }
gfCNCPoint2[10225] = {X 166.5856, Y 9.9932, Z -3.0000, A 0.000, B 0.000, C 0.000 }
gfCNCPoint2[10226] = {X 166.6021, Y 10.4835, Z -3.0000, A 0.000, B 0.000, C 0.000 }
gfCNCPoint2[10227] = {X 166.6021, Y 13.0969, Z -3.0000, A 0.000, B 0.000, C 0.000 }
gfCNCPoint2[10228] = {X 166.8569, Y 11.8210, Z -3.0000, A 0.000, B 0.000, C 0.000 }
gfCNCPoint2[10229] = {X 167.3348, Y 10.6108, Z -3.0000, A 0.000, B 0.000, C 0.000 }
gfCNCPoint2[10230] = {X 168.0205, Y 9.5050, Z -3.0000, A 0.000, B 0.000, C 0.000 }
gfCNCPoint2[10231] = {X 168.0205, Y 7.1050, Z -3.0000, A 0.000, B 0.000, C 0.000 }
gfCNCPoint2[10232] = {X 162.8435, Y 7.1050, Z -3.0000, A 0.000, B 0.000, C 0.000 }
gfCNCPoint2[10233] = {X 163.4703, Y 7.9132, Z -3.0000, A 0.000, B 0.000, C 0.000 }
gfCNCPoint2[10234] = {X 163.9149, Y 8.8342, Z -3.0000, A 0.000, B 0.000, C 0.000 }
gfCNCPoint2[10235] = {X 164.1578, Y 9.8276, Z -3.0000, A 0.000, B 0.000, C 0.000 }
gfCNCPoint2[10236] = {X 164.1910, Y 10.1548, Z -3.0000, A 0.000, B 0.000, C 0.000 }
gfCNCPoint2[10237] = {X 164.2021, Y 10.4835, Z -3.0000, A 0.000, B 0.000, C 0.000 }
gfCNCPoint2[10238] = {X 164.2021, Y 17.4615, Z -3.0000, A 0.000, B 0.000, C 0.000 }
gfCNCPoint2[10239] = {X 164.1139, Y 18.3848, Z -3.0000, A 0.000, B 0.000, C 0.000 }
gfCNCPoint2[10240] = {X 163.8527, Y 19.2747, Z -3.0000, A 0.000, B 0.000, C 0.000 }
gfCNCPoint2[10241] = {X 163.4279, Y 20.0991, Z -3.0000, A 0.000, B 0.000, C 0.000 }
gfCNCPoint2[10242] = {X 162.8547, Y 20.8283, Z -3.0000, A 0.000, B 0.000, C 0.000 }
gfCNCPoint2[10243] = {X 162.1539, Y 21.4358, Z -3.0000, A 0.000, B 0.000, C 0.000 }
gfCNCPoint2[10244] = {X 161.3509, Y 21.8998, Z -3.0000, A 0.000, B 0.000, C 0.000 }
gfCNCPoint2[10245] = {X 160.4745, Y 22.2035, Z -3.0000, A 0.000, B 0.000, C 0.000 }
gfCNCPoint2[10246] = {X 162.1749, Y 29.1999, Z -3.0000, A 0.000, B 0.000, C 0.000 }
gfCNCPoint2[10247] = {X 161.1123, Y 29.4082, Z -3.0000, A 0.000, B 0.000, C 0.000 }
gfCNCPoint2[10248] = {X 160.0353, Y 29.5205, Z -3.0000, A 0.000, B 0.000, C 0.000 }
gfCNCPoint2[10249] = {X 160.0346, Y 38.3366, Z -3.0000, A 0.000, B 0.000, C 0.000 }
gfCNCPoint2[10250] = {X 160.6828, Y 39.6937, Z -3.0000, A 0.000, B 0.000, C 0.000 }
gfCNCPoint2[10251] = {X 161.1579, Y 41.1206, Z -3.0000, A 0.000, B 0.000, C 0.000 }
gfCNCPoint2[10252] = {X 162.0484, Y 41.1205, Z -3.0000, A 0.000, B 0.000, C 0.000 }
gfCNCPoint2[10253] = {X 161.6741, Y 39.3710, Z -3.0000, A 0.000, B 0.000, C 0.000 }
gfCNCPoint2[10254] = {X 161.4501, Y 37.5959, Z -3.0000, A 0.000, B 0.000, C 0.000 }
gfCNCPoint2[10255] = {X 161.3318, Y 35.4806, Z -3.0000, A 0.000, B 0.000, C 0.000 }
gfCNCPoint2[10256] = {X 161.4140, Y 33.3635, Z -3.0000, A 0.000, B 0.000, C 0.000 }
gfCNCPoint2[10257] = {X 161.6958, Y 31.2637, Z -3.0000, A 0.000, B 0.000, C 0.000 }
gfCNCPoint2[10258] = {X 162.1749, Y 29.1999, Z -3.0000, A 0.000, B 0.000, C 0.000 }
gfCNCPoint2[10259] = {X 161.6081, Y 26.8677, Z -3.0000, A 0.000, B 0.000, C 0.000 }
gfCNCPoint2[10260] = {X 160.4733, Y 27.0728, Z -3.0000, A 0.000, B 0.000, C 0.000 }
gfCNCPoint2[10261] = {X 159.3221, Y 27.1415, Z -3.0000, A 0.000, B 0.000, C 0.000 }
gfCNCPoint2[10262] = {X 158.6539, Y 27.1415, Z -3.0000, A 0.000, B 0.000, C 0.000 }
gfCNCPoint2[10263] = {X 158.1439, Y 27.1257, Z -3.0000, A 0.000, B 0.000, C 0.000 }
gfCNCPoint2[10264] = {X 157.6355, Y 27.0832, Z -3.0000, A 0.000, B 0.000, C 0.000 }
gfCNCPoint2[10265] = {X 157.6346, Y 38.9961, Z -3.0000, A 0.000, B 0.000, C 0.000 }
gfCNCPoint2[10266] = {X 158.2184, Y 40.0484, Z -3.0000, A 0.000, B 0.000, C 0.000 }
gfCNCPoint2[10267] = {X 158.6678, Y 41.1649, Z -3.0000, A 0.000, B 0.000, C 0.000 }
gfCNCPoint2[10268] = {X 158.9756, Y 42.3283, Z -3.0000, A 0.000, B 0.000, C 0.000 }
gfCNCPoint2[10269] = {X 159.1374, Y 43.5209, Z -3.0000, A 0.000, B 0.000, C 0.000 }
gfCNCPoint2[10270] = {X 165.4302, Y 43.5200, Z -3.0000, A 0.000, B 0.000, C 0.000 }
gfCNCPoint2[10271] = {X 164.8367, Y 42.0421, Z -3.0000, A 0.000, B 0.000, C 0.000 }
gfCNCPoint2[10272] = {X 164.3718, Y 40.5188, Z -3.0000, A 0.000, B 0.000, C 0.000 }
gfCNCPoint2[10273] = {X 164.0382, Y 38.9573, Z -3.0000, A 0.000, B 0.000, C 0.000 }
gfCNCPoint2[10274] = {X 163.8399, Y 37.3730, Z -3.0000, A 0.000, B 0.000, C 0.000 }
gfCNCPoint2[10275] = {X 163.7319, Y 35.4784, Z -3.0000, A 0.000, B 0.000, C 0.000 }
gfCNCPoint2[10276] = {X 163.8041, Y 33.5820, Z -3.0000, A 0.000, B 0.000, C 0.000 }
gfCNCPoint2[10277] = {X 164.0557, Y 31.7011, Z -3.0000, A 0.000, B 0.000, C 0.000 }
gfCNCPoint2[10278] = {X 164.4844, Y 29.8525, Z -3.0000, A 0.000, B 0.000, C 0.000 }
gfCNCPoint2[10279] = {X 164.8364, Y 28.7333, Z -3.0000, A 0.000, B 0.000, C 0.000 }
gfCNCPoint2[10280] = {X 165.2535, Y 27.6368, Z -3.0000, A 0.000, B 0.000, C 0.000 }
gfCNCPoint2[10281] = {X 165.8701, Y 26.3060, Z -3.0000, A 0.000, B 0.000, C 0.000 }
gfCNCPoint2[10282] = {X 166.6044, Y 25.0364, Z -3.0000, A 0.000, B 0.000, C 0.000 }
gfCNCPoint2[10283] = {X 167.4504, Y 23.8382, Z -3.0000, A 0.000, B 0.000, C 0.000 }
gfCNCPoint2[10284] = {X 167.1640, Y 23.1367, Z -3.0000, A 0.000, B 0.000, C 0.000 }
gfCNCPoint2[10285] = {X 166.2873, Y 24.1837, Z -3.0000, A 0.000, B 0.000, C 0.000 }
gfCNCPoint2[10286] = {X 165.2721, Y 25.0970, Z -3.0000, A 0.000, B 0.000, C 0.000 }
gfCNCPoint2[10287] = {X 164.1385, Y 25.8583, Z -3.0000, A 0.000, B 0.000, C 0.000 }
gfCNCPoint2[10288] = {X 162.9090, Y 26.4525, Z -3.0000, A 0.000, B 0.000, C 0.000 }
gfCNCPoint2[10289] = {X 161.6081, Y 26.8677, Z -3.0000, A 0.000, B 0.000, C 0.000 }
gfCNCPoint2[10290] = {X 161.0413, Y 24.5356, Z -3.0000, A 0.000, B 0.000, C 0.000 }
gfCNCPoint2[10291] = {X 160.1878, Y 24.6899, Z -3.0000, A 0.000, B 0.000, C 0.000 }
gfCNCPoint2[10292] = {X 159.3221, Y 24.7415, Z -3.0000, A 0.000, B 0.000, C 0.000 }
gfCNCPoint2[10293] = {X 158.6652, Y 24.7415, Z -3.0000, A 0.000, B 0.000, C 0.000 }
gfCNCPoint2[10294] = {X 158.2811, Y 24.7296, Z -3.0000, A 0.000, B 0.000, C 0.000 }
gfCNCPoint2[10295] = {X 157.8982, Y 24.6976, Z -3.0000, A 0.000, B 0.000, C 0.000 }
gfCNCPoint2[10296] = {X 156.9778, Y 24.5362, Z -3.0000, A 0.000, B 0.000, C 0.000 }
gfCNCPoint2[10297] = {X 156.0854, Y 24.2588, Z -3.0000, A 0.000, B 0.000, C 0.000 }
gfCNCPoint2[10298] = {X 155.2357, Y 23.8699, Z -3.0000, A 0.000, B 0.000, C 0.000 }
gfCNCPoint2[10299] = {X 155.2345, Y 39.7517, Z -3.0000, A 0.000, B 0.000, C 0.000 }
gfCNCPoint2[10300] = {X 155.8253, Y 40.6438, Z -3.0000, A 0.000, B 0.000, C 0.000 }
gfCNCPoint2[10301] = {X 156.2797, Y 41.6124, Z -3.0000, A 0.000, B 0.000, C 0.000 }
gfCNCPoint2[10302] = {X 156.5881, Y 42.6370, Z -3.0000, A 0.000, B 0.000, C 0.000 }
gfCNCPoint2[10303] = {X 156.7437, Y 43.6955, Z -3.0000, A 0.000, B 0.000, C 0.000 }
gfCNCPoint2[10304] = {X 156.7578, Y 43.9473, Z -3.0000, A 0.000, B 0.000, C 0.000 }
gfCNCPoint2[10305] = {X 156.7631, Y 44.1994, Z -3.0000, A 0.000, B 0.000, C 0.000 }
gfCNCPoint2[10306] = {X 156.7629, Y 45.0587, Z -3.0000, A 0.000, B 0.000, C 0.000 }
gfCNCPoint2[10307] = {X 156.7352, Y 45.6370, Z -3.0000, A 0.000, B 0.000, C 0.000 }
gfCNCPoint2[10308] = {X 156.6616, Y 46.2112, Z -3.0000, A 0.000, B 0.000, C 0.000 }
gfCNCPoint2[10309] = {X 157.9052, Y 46.0006, Z -3.0000, A 0.000, B 0.000, C 0.000 }
gfCNCPoint2[10310] = {X 159.1640, Y 45.9207, Z -3.0000, A 0.000, B 0.000, C 0.000 }
gfCNCPoint2[10311] = {X 159.2310, Y 45.9202, Z -3.0000, A 0.000, B 0.000, C 0.000 }
gfCNCPoint2[10312] = {X 159.2980, Y 45.9200, Z -3.0000, A 0.000, B 0.000, C 0.000 }
gfCNCPoint2[10313] = {X 169.6836, Y 45.9200, Z -3.0000, A 0.000, B 0.000, C 0.000 }
gfCNCPoint2[10314] = {X 168.9029, Y 44.8481, Z -3.0000, A 0.000, B 0.000, C 0.000 }
gfCNCPoint2[10315] = {X 168.2124, Y 43.7159, Z -3.0000, A 0.000, B 0.000, C 0.000 }
gfCNCPoint2[10316] = {X 167.6170, Y 42.5310, Z -3.0000, A 0.000, B 0.000, C 0.000 }
gfCNCPoint2[10317] = {X 166.9490, Y 40.7946, Z -3.0000, A 0.000, B 0.000, C 0.000 }
gfCNCPoint2[10318] = {X 166.4845, Y 38.9931, Z -3.0000, A 0.000, B 0.000, C 0.000 }
gfCNCPoint2[10319] = {X 166.2297, Y 37.1502, Z -3.0000, A 0.000, B 0.000, C 0.000 }
gfCNCPoint2[10320] = {X 166.1314, Y 35.3978, Z -3.0000, A 0.000, B 0.000, C 0.000 }
gfCNCPoint2[10321] = {X 166.2081, Y 33.6443, Z -3.0000, A 0.000, B 0.000, C 0.000 }
gfCNCPoint2[10322] = {X 166.4592, Y 31.9071, Z -3.0000, A 0.000, B 0.000, C 0.000 }
gfCNCPoint2[10323] = {X 166.8821, Y 30.2037, Z -3.0000, A 0.000, B 0.000, C 0.000 }
gfCNCPoint2[10324] = {X 167.4726, Y 28.5508, Z -3.0000, A 0.000, B 0.000, C 0.000 }
gfCNCPoint2[10325] = {X 168.2334, Y 26.9816, Z -3.0000, A 0.000, B 0.000, C 0.000 }
gfCNCPoint2[10326] = {X 169.1858, Y 25.5207, Z -3.0000, A 0.000, B 0.000, C 0.000 }
gfCNCPoint2[10327] = {X 170.3146, Y 24.1914, Z -3.0000, A 0.000, B 0.000, C 0.000 }
gfCNCPoint2[10328] = {X 169.9866, Y 23.6225, Z -3.0000, A 0.000, B 0.000, C 0.000 }
gfCNCPoint2[10329] = {X 169.7112, Y 23.0264, Z -3.0000, A 0.000, B 0.000, C 0.000 }
gfCNCPoint2[10330] = {X 167.1001, Y 16.6309, Z -3.0000, A 0.000, B 0.000, C 0.000 }
gfCNCPoint2[10331] = {X 166.7820, Y 15.6636, Z -3.0000, A 0.000, B 0.000, C 0.000 }
gfCNCPoint2[10332] = {X 166.6021, Y 14.6613, Z -3.0000, A 0.000, B 0.000, C 0.000 }
gfCNCPoint2[10333] = {X 166.6021, Y 17.4615, Z -3.0000, A 0.000, B 0.000, C 0.000 }
gfCNCPoint2[10334] = {X 166.5130, Y 18.5970, Z -3.0000, A 0.000, B 0.000, C 0.000 }
gfCNCPoint2[10335] = {X 166.2479, Y 19.7047, Z -3.0000, A 0.000, B 0.000, C 0.000 }
gfCNCPoint2[10336] = {X 165.8132, Y 20.7575, Z -3.0000, A 0.000, B 0.000, C 0.000 }
gfCNCPoint2[10337] = {X 165.2197, Y 21.7296, Z -3.0000, A 0.000, B 0.000, C 0.000 }
gfCNCPoint2[10338] = {X 164.3787, Y 22.6988, Z -3.0000, A 0.000, B 0.000, C 0.000 }
gfCNCPoint2[10339] = {X 163.3807, Y 23.5052, Z -3.0000, A 0.000, B 0.000, C 0.000 }
gfCNCPoint2[10340] = {X 162.2566, Y 24.1239, Z -3.0000, A 0.000, B 0.000, C 0.000 }
gfCNCPoint2[10341] = {X 161.0413, Y 24.5356, Z -3.0000, A 0.000, B 0.000, C 0.000 }
gfCNCPoint2[10342] = {X 160.4745, Y 22.2035, Z -3.0000, A 0.000, B 0.000, C 0.000 }
gfCNCPoint2[10343] = {X 159.9024, Y 22.3069, Z -3.0000, A 0.000, B 0.000, C 0.000 }
gfCNCPoint2[10344] = {X 159.3221, Y 22.3415, Z -3.0000, A 0.000, B 0.000, C 0.000 }
gfCNCPoint2[10345] = {X 158.6764, Y 22.3415, Z -3.0000, A 0.000, B 0.000, C 0.000 }
gfCNCPoint2[10346] = {X 157.8797, Y 22.2728, Z -3.0000, A 0.000, B 0.000, C 0.000 }
gfCNCPoint2[10347] = {X 157.1046, Y 22.0758, Z -3.0000, A 0.000, B 0.000, C 0.000 }
gfCNCPoint2[10348] = {X 156.3717, Y 21.7558, Z -3.0000, A 0.000, B 0.000, C 0.000 }
gfCNCPoint2[10349] = {X 155.5229, Y 21.1779, Z -3.0000, A 0.000, B 0.000, C 0.000 }
gfCNCPoint2[10350] = {X 154.8126, Y 20.4364, Z -3.0000, A 0.000, B 0.000, C 0.000 }
gfCNCPoint2[10351] = {X 152.8359, Y 20.4374, Z -3.0000, A 0.000, B 0.000, C 0.000 }
gfCNCPoint2[10352] = {X 152.8345, Y 40.6542, Z -3.0000, A 0.000, B 0.000, C 0.000 }
gfCNCPoint2[10353] = {X 153.1755, Y 41.0230, Z -3.0000, A 0.000, B 0.000, C 0.000 }
gfCNCPoint2[10354] = {X 153.6796, Y 41.7268, Z -3.0000, A 0.000, B 0.000, C 0.000 }
gfCNCPoint2[10355] = {X 154.0526, Y 42.5082, Z -3.0000, A 0.000, B 0.000, C 0.000 }
gfCNCPoint2[10356] = {X 154.2828, Y 43.3428, Z -3.0000, A 0.000, B 0.000, C 0.000 }
gfCNCPoint2[10357] = {X 154.3631, Y 44.2048, Z -3.0000, A 0.000, B 0.000, C 0.000 }
gfCNCPoint2[10358] = {X 154.3629, Y 45.0469, Z -3.0000, A 0.000, B 0.000, C 0.000 }
gfCNCPoint2[10359] = {X 154.3441, Y 45.4307, Z -3.0000, A 0.000, B 0.000, C 0.000 }
gfCNCPoint2[10360] = {X 154.2951, Y 45.8119, Z -3.0000, A 0.000, B 0.000, C 0.000 }
gfCNCPoint2[10361] = {X 154.0370, Y 46.7541, Z -3.0000, A 0.000, B 0.000, C 0.000 }
gfCNCPoint2[10362] = {X 153.5963, Y 47.6260, Z -3.0000, A 0.000, B 0.000, C 0.000 }
gfCNCPoint2[10363] = {X 152.9909, Y 48.3926, Z -3.0000, A 0.000, B 0.000, C 0.000 }
gfCNCPoint2[10364] = {X 152.2448, Y 49.0233, Z -3.0000, A 0.000, B 0.000, C 0.000 }
gfCNCPoint2[10365] = {X 151.3881, Y 49.4928, Z -3.0000, A 0.000, B 0.000, C 0.000 }
gfCNCPoint2[10366] = {X 150.4551, Y 49.7822, Z -3.0000, A 0.000, B 0.000, C 0.000 }
gfCNCPoint2[10367] = {X 149.4831, Y 49.8800, Z -3.0000, A 0.000, B 0.000, C 0.000 }
gfCNCPoint2[10368] = {X 143.0396, Y 49.8800, Z -3.0000, A 0.000, B 0.000, C 0.000 }
gfCNCPoint2[10369] = {X 142.0923, Y 49.7872, Z -3.0000, A 0.000, B 0.000, C 0.000 }
gfCNCPoint2[10370] = {X 141.1811, Y 49.5122, Z -3.0000, A 0.000, B 0.000, C 0.000 }
gfCNCPoint2[10371] = {X 140.3405, Y 49.0656, Z -3.0000, A 0.000, B 0.000, C 0.000 }
gfCNCPoint2[10372] = {X 139.6026, Y 48.4643, Z -3.0000, A 0.000, B 0.000, C 0.000 }
gfCNCPoint2[10373] = {X 138.9955, Y 47.7312, Z -3.0000, A 0.000, B 0.000, C 0.000 }
gfCNCPoint2[10374] = {X 138.5423, Y 46.8942, Z -3.0000, A 0.000, B 0.000, C 0.000 }
gfCNCPoint2[10375] = {X 138.2601, Y 45.9852, Z -3.0000, A 0.000, B 0.000, C 0.000 }
gfCNCPoint2[10376] = {X 138.1598, Y 45.0386, Z -3.0000, A 0.000, B 0.000, C 0.000 }
gfCNCPoint2[10377] = {X 138.1601, Y 44.1417, Z -3.0000, A 0.000, B 0.000, C 0.000 }
gfCNCPoint2[10378] = {X 138.2148, Y 43.4769, Z -3.0000, A 0.000, B 0.000, C 0.000 }
gfCNCPoint2[10379] = {X 138.3597, Y 42.8258, Z -3.0000, A 0.000, B 0.000, C 0.000 }
gfCNCPoint2[10380] = {X 129.1532, Y 40.1052, Z -3.0000, A 0.000, B 0.000, C 0.000 }
gfCNCPoint2[10381] = {X 129.5665, Y 38.9035, Z -3.0000, A 0.000, B 0.000, C 0.000 }
gfCNCPoint2[10382] = {X 130.0836, Y 37.7426, Z -3.0000, A 0.000, B 0.000, C 0.000 }
gfCNCPoint2[10383] = {X 130.0836, Y 31.6021, Z -3.0000, A 0.000, B 0.000, C 0.000 }
gfCNCPoint2[10384] = {X 129.2060, Y 31.3796, Z -3.0000, A 0.000, B 0.000, C 0.000 }
gfCNCPoint2[10385] = {X 128.3439, Y 31.1028, Z -3.0000, A 0.000, B 0.000, C 0.000 }
gfCNCPoint2[10386] = {X 128.3436, Y 38.3282, Z -3.0000, A 0.000, B 0.000, C 0.000 }
gfCNCPoint2[10387] = {X 128.7844, Y 39.2003, Z -3.0000, A 0.000, B 0.000, C 0.000 }
gfCNCPoint2[10388] = {X 129.1532, Y 40.1052, Z -3.0000, A 0.000, B 0.000, C 0.000 }
gfCNCPoint2[10389] = {X 131.4548, Y 40.7854, Z -3.0000, A 0.000, B 0.000, C 0.000 }
gfCNCPoint2[10390] = {X 131.9017, Y 39.5320, Z -3.0000, A 0.000, B 0.000, C 0.000 }
gfCNCPoint2[10391] = {X 132.4836, Y 38.3354, Z -3.0000, A 0.000, B 0.000, C 0.000 }
gfCNCPoint2[10392] = {X 132.4836, Y 29.5202, Z -3.0000, A 0.000, B 0.000, C 0.000 }
gfCNCPoint2[10393] = {X 131.3524, Y 29.3993, Z -3.0000, A 0.000, B 0.000, C 0.000 }
gfCNCPoint2[10394] = {X 130.2375, Y 29.1725, Z -3.0000, A 0.000, B 0.000, C 0.000 }
gfCNCPoint2[10395] = {X 129.1489, Y 28.8418, Z -3.0000, A 0.000, B 0.000, C 0.000 }
gfCNCPoint2[10396] = {X 128.0245, Y 28.3764, Z -3.0000, A 0.000, B 0.000, C 0.000 }
gfCNCPoint2[10397] = {X 126.9526, Y 27.8002, Z -3.0000, A 0.000, B 0.000, C 0.000 }
gfCNCPoint2[10398] = {X 125.9441, Y 27.1192, Z -3.0000, A 0.000, B 0.000, C 0.000 }
gfCNCPoint2[10399] = {X 125.9435, Y 38.9888, Z -3.0000, A 0.000, B 0.000, C 0.000 }
gfCNCPoint2[10400] = {X 126.4736, Y 39.9281, Z -3.0000, A 0.000, B 0.000, C 0.000 }
gfCNCPoint2[10401] = {X 126.8960, Y 40.9205, Z -3.0000, A 0.000, B 0.000, C 0.000 }
gfCNCPoint2[10402] = {X 127.2098, Y 41.9730, Z -3.0000, A 0.000, B 0.000, C 0.000 }
gfCNCPoint2[10403] = {X 127.4025, Y 43.0542, Z -3.0000, A 0.000, B 0.000, C 0.000 }
gfCNCPoint2[10404] = {X 127.4714, Y 44.1502, Z -3.0000, A 0.000, B 0.000, C 0.000 }
gfCNCPoint2[10405] = {X 127.4716, Y 45.0000, Z -3.0000, A 0.000, B 0.000, C 0.000 }
gfCNCPoint2[10406] = {X 127.4070, Y 46.1159, Z -3.0000, A 0.000, B 0.000, C 0.000 }
gfCNCPoint2[10407] = {X 127.2143, Y 47.2168, Z -3.0000, A 0.000, B 0.000, C 0.000 }
gfCNCPoint2[10408] = {X 126.8960, Y 48.2883, Z -3.0000, A 0.000, B 0.000, C 0.000 }
gfCNCPoint2[10409] = {X 126.2883, Y 49.6376, Z -3.0000, A 0.000, B 0.000, C 0.000 }
gfCNCPoint2[10410] = {X 125.4821, Y 50.8786, Z -3.0000, A 0.000, B 0.000, C 0.000 }
gfCNCPoint2[10411] = {X 124.4962, Y 51.9821, Z -3.0000, A 0.000, B 0.000, C 0.000 }
gfCNCPoint2[10412] = {X 123.3536, Y 52.9225, Z -3.0000, A 0.000, B 0.000, C 0.000 }
gfCNCPoint2[10413] = {X 122.0810, Y 53.6778, Z -3.0000, A 0.000, B 0.000, C 0.000 }
gfCNCPoint2[10414] = {X 120.7081, Y 54.2302, Z -3.0000, A 0.000, B 0.000, C 0.000 }
gfCNCPoint2[10415] = {X 119.2671, Y 54.5669, Z -3.0000, A 0.000, B 0.000, C 0.000 }
gfCNCPoint2[10416] = {X 117.7916, Y 54.6800, Z -3.0000, A 0.000, B 0.000, C 0.000 }
gfCNCPoint2[10417] = {X 111.9185, Y 54.6800, Z -3.0000, A 0.000, B 0.000, C 0.000 }
gfCNCPoint2[10418] = {X 110.6386, Y 54.5950, Z -3.0000, A 0.000, B 0.000, C 0.000 }
gfCNCPoint2[10419] = {X 109.3812, Y 54.3415, Z -3.0000, A 0.000, B 0.000, C 0.000 }
gfCNCPoint2[10420] = {X 108.1683, Y 53.9240, Z -3.0000, A 0.000, B 0.000, C 0.000 }
gfCNCPoint2[10421] = {X 107.0213, Y 53.3498, Z -3.0000, A 0.000, B 0.000, C 0.000 }
gfCNCPoint2[10422] = {X 106.6480, Y 53.5578, Z -3.0000, A 0.000, B 0.000, C 0.000 }
gfCNCPoint2[10423] = {X 106.2658, Y 53.7492, Z -3.0000, A 0.000, B 0.000, C 0.000 }
gfCNCPoint2[10424] = {X 105.0149, Y 54.2383, Z -3.0000, A 0.000, B 0.000, C 0.000 }
gfCNCPoint2[10425] = {X 103.7084, Y 54.5495, Z -3.0000, A 0.000, B 0.000, C 0.000 }
gfCNCPoint2[10426] = {X 102.3713, Y 54.6768, Z -3.0000, A 0.000, B 0.000, C 0.000 }
gfCNCPoint2[10427] = {X 101.0295, Y 54.6179, Z -3.0000, A 0.000, B 0.000, C 0.000 }
gfCNCPoint2[10428] = {X 99.7088, Y 54.3738, Z -3.0000, A 0.000, B 0.000, C 0.000 }
gfCNCPoint2[10429] = {X 98.4345, Y 53.9493, Z -3.0000, A 0.000, B 0.000, C 0.000 }
gfCNCPoint2[10430] = {X 97.2313, Y 53.3524, Z -3.0000, A 0.000, B 0.000, C 0.000 }
gfCNCPoint2[10431] = {X 96.0852, Y 53.9255, Z -3.0000, A 0.000, B 0.000, C 0.000 }
gfCNCPoint2[10432] = {X 94.8734, Y 54.3422, Z -3.0000, A 0.000, B 0.000, C 0.000 }
gfCNCPoint2[10433] = {X 93.6172, Y 54.5952, Z -3.0000, A 0.000, B 0.000, C 0.000 }
gfCNCPoint2[10434] = {X 92.3385, Y 54.6800, Z -3.0000, A 0.000, B 0.000, C 0.000 }
gfCNCPoint2[10435] = {X 85.8951, Y 54.6800, Z -3.0000, A 0.000, B 0.000, C 0.000 }
gfCNCPoint2[10436] = {X 84.6159, Y 54.5951, Z -3.0000, A 0.000, B 0.000, C 0.000 }
gfCNCPoint2[10437] = {X 83.3592, Y 54.3419, Z -3.0000, A 0.000, B 0.000, C 0.000 }
gfCNCPoint2[10438] = {X 82.1469, Y 53.9249, Z -3.0000, A 0.000, B 0.000, C 0.000 }
gfCNCPoint2[10439] = {X 81.0644, Y 55.1572, Z -3.0000, A 0.000, B 0.000, C 0.000 }
gfCNCPoint2[10440] = {X 79.8495, Y 56.2591, Z -3.0000, A 0.000, B 0.000, C 0.000 }
gfCNCPoint2[10441] = {X 78.5178, Y 57.2166, Z -3.0000, A 0.000, B 0.000, C 0.000 }
gfCNCPoint2[10442] = {X 77.0863, Y 58.0174, Z -3.0000, A 0.000, B 0.000, C 0.000 }
gfCNCPoint2[10443] = {X 75.5734, Y 58.6511, Z -3.0000, A 0.000, B 0.000, C 0.000 }
gfCNCPoint2[10444] = {X 73.9986, Y 59.1096, Z -3.0000, A 0.000, B 0.000, C 0.000 }
gfCNCPoint2[10445] = {X 72.3820, Y 59.3871, Z -3.0000, A 0.000, B 0.000, C 0.000 }
gfCNCPoint2[10446] = {X 70.7445, Y 59.4800, Z -3.0000, A 0.000, B 0.000, C 0.000 }
gfCNCPoint2[10447] = {X 64.1851, Y 59.4800, Z -3.0000, A 0.000, B 0.000, C 0.000 }
gfCNCPoint2[10448] = {X 62.4203, Y 59.3720, Z -3.0000, A 0.000, B 0.000, C 0.000 }
gfCNCPoint2[10449] = {X 60.6818, Y 59.0498, Z -3.0000, A 0.000, B 0.000, C 0.000 }
gfCNCPoint2[10450] = {X 58.9955, Y 58.5181, Z -3.0000, A 0.000, B 0.000, C 0.000 }
gfCNCPoint2[10451] = {X 57.3866, Y 57.7848, Z -3.0000, A 0.000, B 0.000, C 0.000 }
gfCNCPoint2[10452] = {X 55.8790, Y 56.8608, Z -3.0000, A 0.000, B 0.000, C 0.000 }
gfCNCPoint2[10453] = {X 54.3715, Y 57.7848, Z -3.0000, A 0.000, B 0.000, C 0.000 }
gfCNCPoint2[10454] = {X 52.7626, Y 58.5181, Z -3.0000, A 0.000, B 0.000, C 0.000 }
gfCNCPoint2[10455] = {X 51.0763, Y 59.0498, Z -3.0000, A 0.000, B 0.000, C 0.000 }
gfCNCPoint2[10456] = {X 49.3378, Y 59.3720, Z -3.0000, A 0.000, B 0.000, C 0.000 }
gfCNCPoint2[10457] = {X 47.5729, Y 59.4800, Z -3.0000, A 0.000, B 0.000, C 0.000 }
gfCNCPoint2[10458] = {X 40.6393, Y 59.4800, Z -3.0000, A 0.000, B 0.000, C 0.000 }
gfCNCPoint2[10459] = {X 38.9795, Y 59.3846, Z -3.0000, A 0.000, B 0.000, C 0.000 }
gfCNCPoint2[10460] = {X 37.3416, Y 59.0995, Z -3.0000, A 0.000, B 0.000, C 0.000 }
gfCNCPoint2[10461] = {X 35.7472, Y 58.6286, Z -3.0000, A 0.000, B 0.000, C 0.000 }
gfCNCPoint2[10462] = {X 34.0335, Y 59.4864, Z -3.0000, A 0.000, B 0.000, C 0.000 }
gfCNCPoint2[10463] = {X 32.2415, Y 60.1654, Z -3.0000, A 0.000, B 0.000, C 0.000 }
gfCNCPoint2[10464] = {X 30.3897, Y 60.6587, Z -3.0000, A 0.000, B 0.000, C 0.000 }
gfCNCPoint2[10465] = {X 28.4973, Y 60.9610, Z -3.0000, A 0.000, B 0.000, C 0.000 }
gfCNCPoint2[10466] = {X 26.8405, Y 61.6571, Z -3.0000, A 0.000, B 0.000, C 0.000 }
gfCNCPoint2[10467] = {X 25.1557, Y 62.2824, Z -3.0000, A 0.000, B 0.000, C 0.000 }
gfCNCPoint2[10468] = {X 22.5109, Y 63.1272, Z -3.0000, A 0.000, B 0.000, C 0.000 }
gfCNCPoint2[10469] = {X 19.8106, Y 63.7730, Z -3.0000, A 0.000, B 0.000, C 0.000 }
gfCNCPoint2[10470] = {X 17.0697, Y 64.2161, Z -3.0000, A 0.000, B 0.000, C 0.000 }
gfCNCPoint2[10471] = {X 14.3035, Y 64.4541, Z -3.0000, A 0.000, B 0.000, C 0.000 }
gfCNCPoint2[10472] = {X 14.3035, Y 85.6950, Z -3.0000, A 0.000, B 0.000, C 0.000 }
gfCNCPoint2[10473] = {X 112.5246, Y 85.6950, Z -3.0000, A 0.000, B 0.000, C 0.000 }
gfCNCPoint2[10474] = {X 113.6274, Y 84.5920, Z -3.0000, A 0.000, B 0.000, C 0.000 }
gfCNCPoint2[10475] = {X 114.8273, Y 83.5956, Z -3.0000, A 0.000, B 0.000, C 0.000 }
gfCNCPoint2[10476] = {X 116.1140, Y 82.7142, Z -3.0000, A 0.000, B 0.000, C 0.000 }
gfCNCPoint2[10477] = {X 117.4766, Y 81.9553, Z -3.0000, A 0.000, B 0.000, C 0.000 }
gfCNCPoint2[10478] = {X 111.0585, Y 69.0646, Z -3.0000, A 0.000, B 0.000, C 0.000 }
gfCNCPoint2[10479] = {X 109.0296, Y 68.9061, Z -3.0000, A 0.000, B 0.000, C 0.000 }
gfCNCPoint2[10480] = {X 107.0213, Y 68.5768, Z -3.0000, A 0.000, B 0.000, C 0.000 }
gfCNCPoint2[10481] = {X 105.0765, Y 68.8983, Z -3.0000, A 0.000, B 0.000, C 0.000 }
gfCNCPoint2[10482] = {X 103.1119, Y 69.0597, Z -3.0000, A 0.000, B 0.000, C 0.000 }
gfCNCPoint2[10483] = {X 101.1407, Y 69.0599, Z -3.0000, A 0.000, B 0.000, C 0.000 }
gfCNCPoint2[10484] = {X 99.1761, Y 68.8989, Z -3.0000, A 0.000, B 0.000, C 0.000 }
gfCNCPoint2[10485] = {X 97.2313, Y 68.5777, Z -3.0000, A 0.000, B 0.000, C 0.000 }
gfCNCPoint2[10486] = {X 95.6131, Y 68.8563, Z -3.0000, A 0.000, B 0.000, C 0.000 }
gfCNCPoint2[10487] = {X 93.9796, Y 69.0240, Z -3.0000, A 0.000, B 0.000, C 0.000 }
gfCNCPoint2[10488] = {X 92.3385, Y 69.0800, Z -3.0000, A 0.000, B 0.000, C 0.000 }
gfCNCPoint2[10489] = {X 86.6884, Y 69.0800, Z -3.0000, A 0.000, B 0.000, C 0.000 }
gfCNCPoint2[10490] = {X 84.7317, Y 70.2668, Z -3.0000, A 0.000, B 0.000, C 0.000 }
gfCNCPoint2[10491] = {X 82.6872, Y 71.2950, Z -3.0000, A 0.000, B 0.000, C 0.000 }
gfCNCPoint2[10492] = {X 107.2716, Y 71.2950, Z -3.0000, A 0.000, B 0.000, C 0.000 }
gfCNCPoint2[10493] = {X 109.1258, Y 70.1132, Z -3.0000, A 0.000, B 0.000, C 0.000 }
gfCNCPoint2[10494] = {X 111.0585, Y 69.0646, Z -3.0000, A 0.000, B 0.000, C 0.000 }
gfCNCPoint2[10495] = {X 112.1282, Y 71.2131, Z -3.0000, A 0.000, B 0.000, C 0.000 }
gfCNCPoint2[10496] = {X 113.1271, Y 70.7394, Z -3.0000, A 0.000, B 0.000, C 0.000 }
gfCNCPoint2[10497] = {X 114.1434, Y 70.3042, Z -3.0000, A 0.000, B 0.000, C 0.000 }
gfCNCPoint2[10498] = {X 117.4437, Y 66.6800, Z -3.0000, A 0.000, B 0.000, C 0.000 }
gfCNCPoint2[10499] = {X 111.9185, Y 66.6800, Z -3.0000, A 0.000, B 0.000, C 0.000 }
gfCNCPoint2[10500] = {X 111.5313, Y 66.6765, Z -3.0000, A 0.000, B 0.000, C 0.000 }
gfCNCPoint2[10501] = {X 111.1442, Y 66.6662, Z -3.0000, A 0.000, B 0.000, C 0.000 }
gfCNCPoint2[10502] = {X 109.0696, Y 66.4920, Z -3.0000, A 0.000, B 0.000, C 0.000 }
gfCNCPoint2[10503] = {X 107.0213, Y 66.1197, Z -3.0000, A 0.000, B 0.000, C 0.000 }
gfCNCPoint2[10504] = {X 105.0796, Y 66.4776, Z -3.0000, A 0.000, B 0.000, C 0.000 }
gfCNCPoint2[10505] = {X 103.1135, Y 66.6574, Z -3.0000, A 0.000, B 0.000, C 0.000 }
gfCNCPoint2[10506] = {X 101.1392, Y 66.6576, Z -3.0000, A 0.000, B 0.000, C 0.000 }
gfCNCPoint2[10507] = {X 99.1730, Y 66.4782, Z -3.0000, A 0.000, B 0.000, C 0.000 }
gfCNCPoint2[10508] = {X 97.2313, Y 66.1207, Z -3.0000, A 0.000, B 0.000, C 0.000 }
gfCNCPoint2[10509] = {X 95.6161, Y 66.4308, Z -3.0000, A 0.000, B 0.000, C 0.000 }
gfCNCPoint2[10510] = {X 93.9821, Y 66.6176, Z -3.0000, A 0.000, B 0.000, C 0.000 }
gfCNCPoint2[10511] = {X 92.3385, Y 66.6800, Z -3.0000, A 0.000, B 0.000, C 0.000 }
gfCNCPoint2[10512] = {X 85.9487, Y 66.6800, Z -3.0000, A 0.000, B 0.000, C 0.000 }
gfCNCPoint2[10513] = {X 83.8780, Y 67.9935, Z -3.0000, A 0.000, B 0.000, C 0.000 }
gfCNCPoint2[10514] = {X 81.6947, Y 69.1098, Z -3.0000, A 0.000, B 0.000, C 0.000 }
gfCNCPoint2[10515] = {X 79.6017, Y 69.9547, Z -3.0000, A 0.000, B 0.000, C 0.000 }
gfCNCPoint2[10516] = {X 77.4443, Y 70.6184, Z -3.0000, A 0.000, B 0.000, C 0.000 }
gfCNCPoint2[10517] = {X 75.2383, Y 71.0959, Z -3.0000, A 0.000, B 0.000, C 0.000 }
gfCNCPoint2[10518] = {X 72.9996, Y 71.3838, Z -3.0000, A 0.000, B 0.000, C 0.000 }
gfCNCPoint2[10519] = {X 70.7445, Y 71.4800, Z -3.0000, A 0.000, B 0.000, C 0.000 }
gfCNCPoint2[10520] = {X 64.1851, Y 71.4800, Z -3.0000, A 0.000, B 0.000, C 0.000 }
gfCNCPoint2[10521] = {X 62.0752, Y 71.3958, Z -3.0000, A 0.000, B 0.000, C 0.000 }
gfCNCPoint2[10522] = {X 59.9787, Y 71.1438, Z -3.0000, A 0.000, B 0.000, C 0.000 }
gfCNCPoint2[10523] = {X 57.9089, Y 70.7255, Z -3.0000, A 0.000, B 0.000, C 0.000 }
gfCNCPoint2[10524] = {X 55.8790, Y 70.1436, Z -3.0000, A 0.000, B 0.000, C 0.000 }
gfCNCPoint2[10525] = {X 53.8492, Y 70.7255, Z -3.0000, A 0.000, B 0.000, C 0.000 }
gfCNCPoint2[10526] = {X 51.7794, Y 71.1438, Z -3.0000, A 0.000, B 0.000, C 0.000 }
gfCNCPoint2[10527] = {X 49.6829, Y 71.3958, Z -3.0000, A 0.000, B 0.000, C 0.000 }
gfCNCPoint2[10528] = {X 47.5729, Y 71.4800, Z -3.0000, A 0.000, B 0.000, C 0.000 }
gfCNCPoint2[10529] = {X 40.6393, Y 71.4800, Z -3.0000, A 0.000, B 0.000, C 0.000 }
gfCNCPoint2[10530] = {X 38.8045, Y 71.4164, Z -3.0000, A 0.000, B 0.000, C 0.000 }
gfCNCPoint2[10531] = {X 36.9785, Y 71.2257, Z -3.0000, A 0.000, B 0.000, C 0.000 }
gfCNCPoint2[10532] = {X 34.3981, Y 72.0346, Z -3.0000, A 0.000, B 0.000, C 0.000 }
gfCNCPoint2[10533] = {X 31.7568, Y 72.6142, Z -3.0000, A 0.000, B 0.000, C 0.000 }
gfCNCPoint2[10534] = {X 30.4650, Y 73.1209, Z -3.0000, A 0.000, B 0.000, C 0.000 }
gfCNCPoint2[10535] = {X 29.1607, Y 73.5945, Z -3.0000, A 0.000, B 0.000, C 0.000 }
gfCNCPoint2[10536] = {X 28.8784, Y 73.6950, Z -3.0000, A 0.000, B 0.000, C 0.000 }
gfCNCPoint2[10537] = {X 108.0338, Y 73.6950, Z -3.0000, A 0.000, B 0.000, C 0.000 }
gfCNCPoint2[10538] = {X 110.0295, Y 72.3690, Z -3.0000, A 0.000, B 0.000, C 0.000 }
gfCNCPoint2[10539] = {X 112.1282, Y 71.2131, Z -3.0000, A 0.000, B 0.000, C 0.000 }
gfCNCPoint2[10540] = {X 113.1979, Y 73.3615, Z -3.0000, A 0.000, B 0.000, C 0.000 }
gfCNCPoint2[10541] = {X 114.3577, Y 72.8186, Z -3.0000, A 0.000, B 0.000, C 0.000 }
gfCNCPoint2[10542] = {X 115.5424, Y 72.3325, Z -3.0000, A 0.000, B 0.000, C 0.000 }
gfCNCPoint2[10543] = {X 123.7283, Y 63.3432, Z -3.0000, A 0.000, B 0.000, C 0.000 }
gfCNCPoint2[10544] = {X 121.7856, Y 63.8618, Z -3.0000, A 0.000, B 0.000, C 0.000 }
gfCNCPoint2[10545] = {X 119.7995, Y 64.1752, Z -3.0000, A 0.000, B 0.000, C 0.000 }
gfCNCPoint2[10546] = {X 117.7916, Y 64.2800, Z -3.0000, A 0.000, B 0.000, C 0.000 }
gfCNCPoint2[10547] = {X 111.9185, Y 64.2800, Z -3.0000, A 0.000, B 0.000, C 0.000 }
gfCNCPoint2[10548] = {X 110.2700, Y 64.2094, Z -3.0000, A 0.000, B 0.000, C 0.000 }
gfCNCPoint2[10549] = {X 108.6336, Y 63.9981, Z -3.0000, A 0.000, B 0.000, C 0.000 }
gfCNCPoint2[10550] = {X 107.0213, Y 63.6477, Z -3.0000, A 0.000, B 0.000, C 0.000 }
gfCNCPoint2[10551] = {X 105.0841, Y 64.0514, Z -3.0000, A 0.000, B 0.000, C 0.000 }
gfCNCPoint2[10552] = {X 103.1158, Y 64.2545, Z -3.0000, A 0.000, B 0.000, C 0.000 }
gfCNCPoint2[10553] = {X 101.1370, Y 64.2547, Z -3.0000, A 0.000, B 0.000, C 0.000 }
gfCNCPoint2[10554] = {X 99.1686, Y 64.0521, Z -3.0000, A 0.000, B 0.000, C 0.000 }
gfCNCPoint2[10555] = {X 97.2313, Y 63.6488, Z -3.0000, A 0.000, B 0.000, C 0.000 }
gfCNCPoint2[10556] = {X 95.6204, Y 63.9986, Z -3.0000, A 0.000, B 0.000, C 0.000 }
gfCNCPoint2[10557] = {X 93.9855, Y 64.2095, Z -3.0000, A 0.000, B 0.000, C 0.000 }
gfCNCPoint2[10558] = {X 92.3385, Y 64.2800, Z -3.0000, A 0.000, B 0.000, C 0.000 }
gfCNCPoint2[10559] = {X 85.8951, Y 64.2800, Z -3.0000, A 0.000, B 0.000, C 0.000 }
gfCNCPoint2[10560] = {X 85.5417, Y 64.2768, Z -3.0000, A 0.000, B 0.000, C 0.000 }
gfCNCPoint2[10561] = {X 85.1884, Y 64.2670, Z -3.0000, A 0.000, B 0.000, C 0.000 }
gfCNCPoint2[10562] = {X 83.3593, Y 65.5113, Z -3.0000, A 0.000, B 0.000, C 0.000 }
gfCNCPoint2[10563] = {X 81.4238, Y 66.5824, Z -3.0000, A 0.000, B 0.000, C 0.000 }
gfCNCPoint2[10564] = {X 79.3981, Y 67.4713, Z -3.0000, A 0.000, B 0.000, C 0.000 }
gfCNCPoint2[10565] = {X 77.2994, Y 68.1706, Z -3.0000, A 0.000, B 0.000, C 0.000 }
gfCNCPoint2[10566] = {X 75.1454, Y 68.6744, Z -3.0000, A 0.000, B 0.000, C 0.000 }
gfCNCPoint2[10567] = {X 72.9543, Y 68.9784, Z -3.0000, A 0.000, B 0.000, C 0.000 }
gfCNCPoint2[10568] = {X 70.7445, Y 69.0800, Z -3.0000, A 0.000, B 0.000, C 0.000 }
gfCNCPoint2[10569] = {X 64.1851, Y 69.0800, Z -3.0000, A 0.000, B 0.000, C 0.000 }
gfCNCPoint2[10570] = {X 62.0678, Y 68.9867, Z -3.0000, A 0.000, B 0.000, C 0.000 }
gfCNCPoint2[10571] = {X 59.9669, Y 68.7076, Z -3.0000, A 0.000, B 0.000, C 0.000 }
gfCNCPoint2[10572] = {X 57.8986, Y 68.2449, Z -3.0000, A 0.000, B 0.000, C 0.000 }
gfCNCPoint2[10573] = {X 55.8790, Y 67.6021, Z -3.0000, A 0.000, B 0.000, C 0.000 }
gfCNCPoint2[10574] = {X 53.8595, Y 68.2449, Z -3.0000, A 0.000, B 0.000, C 0.000 }
gfCNCPoint2[10575] = {X 51.7912, Y 68.7076, Z -3.0000, A 0.000, B 0.000, C 0.000 }
gfCNCPoint2[10576] = {X 49.6903, Y 68.9867, Z -3.0000, A 0.000, B 0.000, C 0.000 }
gfCNCPoint2[10577] = {X 47.5729, Y 69.0800, Z -3.0000, A 0.000, B 0.000, C 0.000 }
gfCNCPoint2[10578] = {X 40.6393, Y 69.0800, Z -3.0000, A 0.000, B 0.000, C 0.000 }
gfCNCPoint2[10579] = {X 38.6741, Y 68.9997, Z -3.0000, A 0.000, B 0.000, C 0.000 }
gfCNCPoint2[10580] = {X 36.7219, Y 68.7592, Z -3.0000, A 0.000, B 0.000, C 0.000 }
gfCNCPoint2[10581] = {X 34.8823, Y 69.3986, Z -3.0000, A 0.000, B 0.000, C 0.000 }
gfCNCPoint2[10582] = {X 33.0031, Y 69.9105, Z -3.0000, A 0.000, B 0.000, C 0.000 }
gfCNCPoint2[10583] = {X 31.0933, Y 70.2924, Z -3.0000, A 0.000, B 0.000, C 0.000 }
gfCNCPoint2[10584] = {X 29.7338, Y 70.8314, Z -3.0000, A 0.000, B 0.000, C 0.000 }
gfCNCPoint2[10585] = {X 28.3598, Y 71.3321, Z -3.0000, A 0.000, B 0.000, C 0.000 }
gfCNCPoint2[10586] = {X 28.2203, Y 71.3820, Z -3.0000, A 0.000, B 0.000, C 0.000 }
gfCNCPoint2[10587] = {X 28.0807, Y 71.4314, Z -3.0000, A 0.000, B 0.000, C 0.000 }
gfCNCPoint2[10588] = {X 26.0067, Y 72.1086, Z -3.0000, A 0.000, B 0.000, C 0.000 }
gfCNCPoint2[10589] = {X 23.9035, Y 72.6885, Z -3.0000, A 0.000, B 0.000, C 0.000 }
gfCNCPoint2[10590] = {X 23.9035, Y 76.0950, Z -3.0000, A 0.000, B 0.000, C 0.000 }
gfCNCPoint2[10591] = {X 108.8319, Y 76.0950, Z -3.0000, A 0.000, B 0.000, C 0.000 }
gfCNCPoint2[10592] = {X 110.2270, Y 75.0899, Z -3.0000, A 0.000, B 0.000, C 0.000 }
gfCNCPoint2[10593] = {X 111.6843, Y 74.1774, Z -3.0000, A 0.000, B 0.000, C 0.000 }
gfCNCPoint2[10594] = {X 113.1979, Y 73.3615, Z -3.0000, A 0.000, B 0.000, C 0.000 }
gfCNCPoint2[10595] = {X 114.2675, Y 75.5099, Z -3.0000, A 0.000, B 0.000, C 0.000 }
gfCNCPoint2[10596] = {X 115.5783, Y 74.9056, Z -3.0000, A 0.000, B 0.000, C 0.000 }
gfCNCPoint2[10597] = {X 116.9230, Y 74.3809, Z -3.0000, A 0.000, B 0.000, C 0.000 }
gfCNCPoint2[10598] = {X 130.4115, Y 59.5687, Z -3.0000, A 0.000, B 0.000, C 0.000 }
gfCNCPoint2[10599] = {X 129.5279, Y 58.7533, Z -3.0000, A 0.000, B 0.000, C 0.000 }
gfCNCPoint2[10600] = {X 128.6970, Y 57.8844, Z -3.0000, A 0.000, B 0.000, C 0.000 }
gfCNCPoint2[10601] = {X 127.3930, Y 58.8833, Z -3.0000, A 0.000, B 0.000, C 0.000 }
gfCNCPoint2[10602] = {X 125.9982, Y 59.7508, Z -3.0000, A 0.000, B 0.000, C 0.000 }
gfCNCPoint2[10603] = {X 124.5256, Y 60.4786, Z -3.0000, A 0.000, B 0.000, C 0.000 }
gfCNCPoint2[10604] = {X 122.9893, Y 61.0598, Z -3.0000, A 0.000, B 0.000, C 0.000 }
gfCNCPoint2[10605] = {X 121.2885, Y 61.5138, Z -3.0000, A 0.000, B 0.000, C 0.000 }
gfCNCPoint2[10606] = {X 119.5496, Y 61.7882, Z -3.0000, A 0.000, B 0.000, C 0.000 }
gfCNCPoint2[10607] = {X 117.7916, Y 61.8800, Z -3.0000, A 0.000, B 0.000, C 0.000 }
gfCNCPoint2[10608] = {X 111.9185, Y 61.8800, Z -3.0000, A 0.000, B 0.000, C 0.000 }
gfCNCPoint2[10609] = {X 110.2649, Y 61.7988, Z -3.0000, A 0.000, B 0.000, C 0.000 }
gfCNCPoint2[10610] = {X 108.6273, Y 61.5560, Z -3.0000, A 0.000, B 0.000, C 0.000 }
gfCNCPoint2[10611] = {X 107.0213, Y 61.1540, Z -3.0000, A 0.000, B 0.000, C 0.000 }
gfCNCPoint2[10612] = {X 105.0907, Y 61.6173, Z -3.0000, A 0.000, B 0.000, C 0.000 }
gfCNCPoint2[10613] = {X 103.1191, Y 61.8506, Z -3.0000, A 0.000, B 0.000, C 0.000 }
gfCNCPoint2[10614] = {X 101.1337, Y 61.8509, Z -3.0000, A 0.000, B 0.000, C 0.000 }
gfCNCPoint2[10615] = {X 99.1620, Y 61.6181, Z -3.0000, A 0.000, B 0.000, C 0.000 }
gfCNCPoint2[10616] = {X 97.2313, Y 61.1553, Z -3.0000, A 0.000, B 0.000, C 0.000 }
gfCNCPoint2[10617] = {X 95.6267, Y 61.5566, Z -3.0000, A 0.000, B 0.000, C 0.000 }
gfCNCPoint2[10618] = {X 93.9906, Y 61.7990, Z -3.0000, A 0.000, B 0.000, C 0.000 }
gfCNCPoint2[10619] = {X 92.3385, Y 61.8800, Z -3.0000, A 0.000, B 0.000, C 0.000 }
gfCNCPoint2[10620] = {X 85.8951, Y 61.8800, Z -3.0000, A 0.000, B 0.000, C 0.000 }
gfCNCPoint2[10621] = {X 85.1609, Y 61.8640, Z -3.0000, A 0.000, B 0.000, C 0.000 }
gfCNCPoint2[10622] = {X 84.4280, Y 61.8161, Z -3.0000, A 0.000, B 0.000, C 0.000 }
gfCNCPoint2[10623] = {X 82.7247, Y 63.0692, Z -3.0000, A 0.000, B 0.000, C 0.000 }
gfCNCPoint2[10624] = {X 80.9073, Y 64.1504, Z -3.0000, A 0.000, B 0.000, C 0.000 }
gfCNCPoint2[10625] = {X 78.9932, Y 65.0494, Z -3.0000, A 0.000, B 0.000, C 0.000 }
gfCNCPoint2[10626] = {X 77.0007, Y 65.7577, Z -3.0000, A 0.000, B 0.000, C 0.000 }
gfCNCPoint2[10627] = {X 74.9487, Y 66.2685, Z -3.0000, A 0.000, B 0.000, C 0.000 }
gfCNCPoint2[10628] = {X 72.8566, Y 66.5769, Z -3.0000, A 0.000, B 0.000, C 0.000 }
gfCNCPoint2[10629] = {X 70.7445, Y 66.6800, Z -3.0000, A 0.000, B 0.000, C 0.000 }
gfCNCPoint2[10630] = {X 64.1851, Y 66.6800, Z -3.0000, A 0.000, B 0.000, C 0.000 }
gfCNCPoint2[10631] = {X 62.0576, Y 66.5754, Z -3.0000, A 0.000, B 0.000, C 0.000 }
gfCNCPoint2[10632] = {X 59.9505, Y 66.2624, Z -3.0000, A 0.000, B 0.000, C 0.000 }
gfCNCPoint2[10633] = {X 57.8844, Y 65.7442, Z -3.0000, A 0.000, B 0.000, C 0.000 }
gfCNCPoint2[10634] = {X 55.8790, Y 65.0258, Z -3.0000, A 0.000, B 0.000, C 0.000 }
gfCNCPoint2[10635] = {X 53.8737, Y 65.7442, Z -3.0000, A 0.000, B 0.000, C 0.000 }
gfCNCPoint2[10636] = {X 51.8075, Y 66.2624, Z -3.0000, A 0.000, B 0.000, C 0.000 }
gfCNCPoint2[10637] = {X 49.7005, Y 66.5754, Z -3.0000, A 0.000, B 0.000, C 0.000 }
gfCNCPoint2[10638] = {X 47.5729, Y 66.6800, Z -3.0000, A 0.000, B 0.000, C 0.000 }
gfCNCPoint2[10639] = {X 40.6393, Y 66.6800, Z -3.0000, A 0.000, B 0.000, C 0.000 }
gfCNCPoint2[10640] = {X 38.5443, Y 66.5785, Z -3.0000, A 0.000, B 0.000, C 0.000 }
gfCNCPoint2[10641] = {X 36.4688, Y 66.2751, Z -3.0000, A 0.000, B 0.000, C 0.000 }
gfCNCPoint2[10642] = {X 34.5050, Y 67.0006, Z -3.0000, A 0.000, B 0.000, C 0.000 }
gfCNCPoint2[10643] = {X 32.4891, Y 67.5658, Z -3.0000, A 0.000, B 0.000, C 0.000 }
gfCNCPoint2[10644] = {X 30.4343, Y 67.9671, Z -3.0000, A 0.000, B 0.000, C 0.000 }
gfCNCPoint2[10645] = {X 29.0051, Y 68.5407, Z -3.0000, A 0.000, B 0.000, C 0.000 }
gfCNCPoint2[10646] = {X 27.5588, Y 69.0696, Z -3.0000, A 0.000, B 0.000, C 0.000 }
gfCNCPoint2[10647] = {X 24.5613, Y 70.0300, Z -3.0000, A 0.000, B 0.000, C 0.000 }
gfCNCPoint2[10648] = {X 21.5035, Y 70.7760, Z -3.0000, A 0.000, B 0.000, C 0.000 }
gfCNCPoint2[10649] = {X 21.5035, Y 78.4950, Z -3.0000, A 0.000, B 0.000, C 0.000 }
gfCNCPoint2[10650] = {X 109.6714, Y 78.4950, Z -3.0000, A 0.000, B 0.000, C 0.000 }
gfCNCPoint2[10651] = {X 111.1263, Y 77.3843, Z -3.0000, A 0.000, B 0.000, C 0.000 }
gfCNCPoint2[10652] = {X 112.6613, Y 76.3874, Z -3.0000, A 0.000, B 0.000, C 0.000 }
gfCNCPoint2[10653] = {X 114.2675, Y 75.5099, Z -3.0000, A 0.000, B 0.000, C 0.000 }
gfCNCPoint2[10654] = {X 115.3372, Y 77.6584, Z -3.0000, A 0.000, B 0.000, C 0.000 }
gfCNCPoint2[10655] = {X 116.7875, Y 77.0016, Z -3.0000, A 0.000, B 0.000, C 0.000 }
gfCNCPoint2[10656] = {X 118.2821, Y 76.4530, Z -3.0000, A 0.000, B 0.000, C 0.000 }
gfCNCPoint2[10657] = {X 133.9637, Y 59.2324, Z -3.0000, A 0.000, B 0.000, C 0.000 }
gfCNCPoint2[10658] = {X 132.7158, Y 58.3549, Z -3.0000, A 0.000, B 0.000, C 0.000 }
gfCNCPoint2[10659] = {X 131.5521, Y 57.3682, Z -3.0000, A 0.000, B 0.000, C 0.000 }
gfCNCPoint2[10660] = {X 130.4824, Y 56.2805, Z -3.0000, A 0.000, B 0.000, C 0.000 }
gfCNCPoint2[10661] = {X 129.6655, Y 55.2988, Z -3.0000, A 0.000, B 0.000, C 0.000 }
gfCNCPoint2[10662] = {X 128.9251, Y 54.2582, Z -3.0000, A 0.000, B 0.000, C 0.000 }
gfCNCPoint2[10663] = {X 128.0750, Y 55.1942, Z -3.0000, A 0.000, B 0.000, C 0.000 }
gfCNCPoint2[10664] = {X 127.1464, Y 56.0525, Z -3.0000, A 0.000, B 0.000, C 0.000 }
gfCNCPoint2[10665] = {X 125.7915, Y 57.0695, Z -3.0000, A 0.000, B 0.000, C 0.000 }
gfCNCPoint2[10666] = {X 124.3270, Y 57.9212, Z -3.0000, A 0.000, B 0.000, C 0.000 }
gfCNCPoint2[10667] = {X 122.7731, Y 58.5961, Z -3.0000, A 0.000, B 0.000, C 0.000 }
gfCNCPoint2[10668] = {X 121.1510, Y 59.0849, Z -3.0000, A 0.000, B 0.000, C 0.000 }
gfCNCPoint2[10669] = {X 119.4828, Y 59.3809, Z -3.0000, A 0.000, B 0.000, C 0.000 }
gfCNCPoint2[10670] = {X 117.7916, Y 59.4800, Z -3.0000, A 0.000, B 0.000, C 0.000 }
gfCNCPoint2[10671] = {X 111.9185, Y 59.4800, Z -3.0000, A 0.000, B 0.000, C 0.000 }
gfCNCPoint2[10672] = {X 110.2569, Y 59.3844, Z -3.0000, A 0.000, B 0.000, C 0.000 }
gfCNCPoint2[10673] = {X 108.6173, Y 59.0987, Z -3.0000, A 0.000, B 0.000, C 0.000 }
gfCNCPoint2[10674] = {X 107.0213, Y 58.6267, Z -3.0000, A 0.000, B 0.000, C 0.000 }
gfCNCPoint2[10675] = {X 105.4260, Y 59.0985, Z -3.0000, A 0.000, B 0.000, C 0.000 }
gfCNCPoint2[10676] = {X 103.7872, Y 59.3842, Z -3.0000, A 0.000, B 0.000, C 0.000 }
gfCNCPoint2[10677] = {X 102.1264, Y 59.4800, Z -3.0000, A 0.000, B 0.000, C 0.000 }
gfCNCPoint2[10678] = {X 100.4656, Y 59.3847, Z -3.0000, A 0.000, B 0.000, C 0.000 }
gfCNCPoint2[10679] = {X 98.8267, Y 59.0996, Z -3.0000, A 0.000, B 0.000, C 0.000 }
gfCNCPoint2[10680] = {X 97.2313, Y 58.6283, Z -3.0000, A 0.000, B 0.000, C 0.000 }
gfCNCPoint2[10681] = {X 95.6367, Y 59.0994, Z -3.0000, A 0.000, B 0.000, C 0.000 }
gfCNCPoint2[10682] = {X 93.9986, Y 59.3845, Z -3.0000, A 0.000, B 0.000, C 0.000 }
gfCNCPoint2[10683] = {X 92.3385, Y 59.4800, Z -3.0000, A 0.000, B 0.000, C 0.000 }
gfCNCPoint2[10684] = {X 85.8951, Y 59.4800, Z -3.0000, A 0.000, B 0.000, C 0.000 }
gfCNCPoint2[10685] = {X 84.7780, Y 59.4368, Z -3.0000, A 0.000, B 0.000, C 0.000 }
gfCNCPoint2[10686] = {X 83.6677, Y 59.3077, Z -3.0000, A 0.000, B 0.000, C 0.000 }
gfCNCPoint2[10687] = {X 82.0978, Y 60.5827, Z -3.0000, A 0.000, B 0.000, C 0.000 }
gfCNCPoint2[10688] = {X 80.4031, Y 61.6862, Z -3.0000, A 0.000, B 0.000, C 0.000 }
gfCNCPoint2[10689] = {X 78.6021, Y 62.6061, Z -3.0000, A 0.000, B 0.000, C 0.000 }
gfCNCPoint2[10690] = {X 76.7146, Y 63.3324, Z -3.0000, A 0.000, B 0.000, C 0.000 }
gfCNCPoint2[10691] = {X 74.7614, Y 63.8569, Z -3.0000, A 0.000, B 0.000, C 0.000 }
gfCNCPoint2[10692] = {X 72.7641, Y 64.1739, Z -3.0000, A 0.000, B 0.000, C 0.000 }
gfCNCPoint2[10693] = {X 70.7445, Y 64.2800, Z -3.0000, A 0.000, B 0.000, C 0.000 }
gfCNCPoint2[10694] = {X 64.1851, Y 64.2800, Z -3.0000, A 0.000, B 0.000, C 0.000 }
gfCNCPoint2[10695] = {X 62.0428, Y 64.1606, Z -3.0000, A 0.000, B 0.000, C 0.000 }
gfCNCPoint2[10696] = {X 59.9269, Y 63.8039, Z -3.0000, A 0.000, B 0.000, C 0.000 }
gfCNCPoint2[10697] = {X 57.8638, Y 63.2143, Z -3.0000, A 0.000, B 0.000, C 0.000 }
gfCNCPoint2[10698] = {X 55.8790, Y 62.3991, Z -3.0000, A 0.000, B 0.000, C 0.000 }
gfCNCPoint2[10699] = {X 53.8942, Y 63.2143, Z -3.0000, A 0.000, B 0.000, C 0.000 }
gfCNCPoint2[10700] = {X 51.8311, Y 63.8039, Z -3.0000, A 0.000, B 0.000, C 0.000 }
gfCNCPoint2[10701] = {X 49.7153, Y 64.1606, Z -3.0000, A 0.000, B 0.000, C 0.000 }
gfCNCPoint2[10702] = {X 47.5729, Y 64.2800, Z -3.0000, A 0.000, B 0.000, C 0.000 }
gfCNCPoint2[10703] = {X 40.6393, Y 64.2800, Z -3.0000, A 0.000, B 0.000, C 0.000 }
gfCNCPoint2[10704] = {X 39.1546, Y 64.2227, Z -3.0000, A 0.000, B 0.000, C 0.000 }
gfCNCPoint2[10705] = {X 37.6787, Y 64.0513, Z -3.0000, A 0.000, B 0.000, C 0.000 }
gfCNCPoint2[10706] = {X 36.2204, Y 63.7668, Z -3.0000, A 0.000, B 0.000, C 0.000 }
gfCNCPoint2[10707] = {X 34.1365, Y 64.5936, Z -3.0000, A 0.000, B 0.000, C 0.000 }
gfCNCPoint2[10708] = {X 31.9836, Y 65.2191, Z -3.0000, A 0.000, B 0.000, C 0.000 }
gfCNCPoint2[10709] = {X 29.7810, Y 65.6376, Z -3.0000, A 0.000, B 0.000, C 0.000 }
gfCNCPoint2[10710] = {X 28.2794, Y 66.2483, Z -3.0000, A 0.000, B 0.000, C 0.000 }
gfCNCPoint2[10711] = {X 26.7578, Y 66.8072, Z -3.0000, A 0.000, B 0.000, C 0.000 }
gfCNCPoint2[10712] = {X 24.2492, Y 67.6229, Z -3.0000, A 0.000, B 0.000, C 0.000 }
gfCNCPoint2[10713] = {X 21.6944, Y 68.2799, Z -3.0000, A 0.000, B 0.000, C 0.000 }
gfCNCPoint2[10714] = {X 19.1035, Y 68.7756, Z -3.0000, A 0.000, B 0.000, C 0.000 }
gfCNCPoint2[10715] = {X 19.1035, Y 80.8950, Z -3.0000, A 0.000, B 0.000, C 0.000 }
gfCNCPoint2[10716] = {X 110.5597, Y 80.8950, Z -3.0000, A 0.000, B 0.000, C 0.000 }
gfCNCPoint2[10717] = {X 112.0540, Y 79.6756, Z -3.0000, A 0.000, B 0.000, C 0.000 }
gfCNCPoint2[10718] = {X 113.6507, Y 78.5939, Z -3.0000, A 0.000, B 0.000, C 0.000 }
gfCNCPoint2[10719] = {X 115.3372, Y 77.6584, Z -3.0000, A 0.000, B 0.000, C 0.000 }
gfCNCPoint2[10720] = {X 116.4069, Y 79.8068, Z -3.0000, A 0.000, B 0.000, C 0.000 }
gfCNCPoint2[10721] = {X 117.9833, Y 79.1081, Z -3.0000, A 0.000, B 0.000, C 0.000 }
gfCNCPoint2[10722] = {X 119.6158, Y 78.5530, Z -3.0000, A 0.000, B 0.000, C 0.000 }
gfCNCPoint2[10723] = {X 137.8576, Y 58.5210, Z -3.0000, A 0.000, B 0.000, C 0.000 }
gfCNCPoint2[10724] = {X 136.5227, Y 57.9306, Z -3.0000, A 0.000, B 0.000, C 0.000 }
gfCNCPoint2[10725] = {X 135.2541, Y 57.2089, Z -3.0000, A 0.000, B 0.000, C 0.000 }
gfCNCPoint2[10726] = {X 134.0101, Y 56.3198, Z -3.0000, A 0.000, B 0.000, C 0.000 }
gfCNCPoint2[10727] = {X 132.8668, Y 55.3045, Z -3.0000, A 0.000, B 0.000, C 0.000 }
gfCNCPoint2[10728] = {X 131.8369, Y 54.1744, Z -3.0000, A 0.000, B 0.000, C 0.000 }
gfCNCPoint2[10729] = {X 130.9319, Y 52.9419, Z -3.0000, A 0.000, B 0.000, C 0.000 }
gfCNCPoint2[10730] = {X 130.2147, Y 51.7225, Z -3.0000, A 0.000, B 0.000, C 0.000 }
gfCNCPoint2[10731] = {X 129.6199, Y 50.4390, Z -3.0000, A 0.000, B 0.000, C 0.000 }
gfCNCPoint2[10732] = {X 129.1532, Y 49.1035, Z -3.0000, A 0.000, B 0.000, C 0.000 }
gfCNCPoint2[10733] = {X 128.6036, Y 50.3877, Z -3.0000, A 0.000, B 0.000, C 0.000 }
gfCNCPoint2[10734] = {X 127.9093, Y 51.5998, Z -3.0000, A 0.000, B 0.000, C 0.000 }
gfCNCPoint2[10735] = {X 127.0798, Y 52.7237, Z -3.0000, A 0.000, B 0.000, C 0.000 }
gfCNCPoint2[10736] = {X 126.0417, Y 53.8239, Z -3.0000, A 0.000, B 0.000, C 0.000 }
gfCNCPoint2[10737] = {X 124.8743, Y 54.7858, Z -3.0000, A 0.000, B 0.000, C 0.000 }
gfCNCPoint2[10738] = {X 123.5958, Y 55.5942, Z -3.0000, A 0.000, B 0.000, C 0.000 }
gfCNCPoint2[10739] = {X 122.2263, Y 56.2365, Z -3.0000, A 0.000, B 0.000, C 0.000 }
gfCNCPoint2[10740] = {X 120.7872, Y 56.7027, Z -3.0000, A 0.000, B 0.000, C 0.000 }
gfCNCPoint2[10741] = {X 119.3012, Y 56.9853, Z -3.0000, A 0.000, B 0.000, C 0.000 }
gfCNCPoint2[10742] = {X 117.7916, Y 57.0800, Z -3.0000, A 0.000, B 0.000, C 0.000 }
gfCNCPoint2[10743] = {X 111.9185, Y 57.0800, Z -3.0000, A 0.000, B 0.000, C 0.000 }
gfCNCPoint2[10744] = {X 110.2431, Y 56.9633, Z -3.0000, A 0.000, B 0.000, C 0.000 }
gfCNCPoint2[10745] = {X 108.6001, Y 56.6153, Z -3.0000, A 0.000, B 0.000, C 0.000 }
gfCNCPoint2[10746] = {X 107.0213, Y 56.0428, Z -3.0000, A 0.000, B 0.000, C 0.000 }
gfCNCPoint2[10747] = {X 105.4432, Y 56.6151, Z -3.0000, A 0.000, B 0.000, C 0.000 }
gfCNCPoint2[10748] = {X 103.8010, Y 56.9630, Z -3.0000, A 0.000, B 0.000, C 0.000 }
gfCNCPoint2[10749] = {X 102.1265, Y 57.0800, Z -3.0000, A 0.000, B 0.000, C 0.000 }
gfCNCPoint2[10750] = {X 100.4519, Y 56.9637, Z -3.0000, A 0.000, B 0.000, C 0.000 }
gfCNCPoint2[10751] = {X 98.8096, Y 56.6164, Z -3.0000, A 0.000, B 0.000, C 0.000 }
gfCNCPoint2[10752] = {X 97.2313, Y 56.0448, Z -3.0000, A 0.000, B 0.000, C 0.000 }
gfCNCPoint2[10753] = {X 95.6538, Y 56.6162, Z -3.0000, A 0.000, B 0.000, C 0.000 }
gfCNCPoint2[10754] = {X 94.0123, Y 56.9635, Z -3.0000, A 0.000, B 0.000, C 0.000 }
gfCNCPoint2[10755] = {X 92.3385, Y 57.0800, Z -3.0000, A 0.000, B 0.000, C 0.000 }
gfCNCPoint2[10756] = {X 85.8951, Y 57.0800, Z -3.0000, A 0.000, B 0.000, C 0.000 }
gfCNCPoint2[10757] = {X 84.3894, Y 56.9858, Z -3.0000, A 0.000, B 0.000, C 0.000 }
gfCNCPoint2[10758] = {X 82.9073, Y 56.7047, Z -3.0000, A 0.000, B 0.000, C 0.000 }
gfCNCPoint2[10759] = {X 81.4846, Y 58.0224, Z -3.0000, A 0.000, B 0.000, C 0.000 }
gfCNCPoint2[10760] = {X 79.9203, Y 59.1682, Z -3.0000, A 0.000, B 0.000, C 0.000 }
gfCNCPoint2[10761] = {X 78.2348, Y 60.1271, Z -3.0000, A 0.000, B 0.000, C 0.000 }
gfCNCPoint2[10762] = {X 76.4504, Y 60.8863, Z -3.0000, A 0.000, B 0.000, C 0.000 }
gfCNCPoint2[10763] = {X 74.5908, Y 61.4359, Z -3.0000, A 0.000, B 0.000, C 0.000 }
gfCNCPoint2[10764] = {X 72.6804, Y 61.7686, Z -3.0000, A 0.000, B 0.000, C 0.000 }
gfCNCPoint2[10765] = {X 70.7445, Y 61.8800, Z -3.0000, A 0.000, B 0.000, C 0.000 }
gfCNCPoint2[10766] = {X 64.1851, Y 61.8800, Z -3.0000, A 0.000, B 0.000, C 0.000 }
gfCNCPoint2[10767] = {X 62.4514, Y 61.7907, Z -3.0000, A 0.000, B 0.000, C 0.000 }
gfCNCPoint2[10768] = {X 60.7359, Y 61.5238, Z -3.0000, A 0.000, B 0.000, C 0.000 }
gfCNCPoint2[10769] = {X 59.0570, Y 61.0822, Z -3.0000, A 0.000, B 0.000, C 0.000 }
gfCNCPoint2[10770] = {X 57.4323, Y 60.4704, Z -3.0000, A 0.000, B 0.000, C 0.000 }
gfCNCPoint2[10771] = {X 55.8790, Y 59.6950, Z -3.0000, A 0.000, B 0.000, C 0.000 }
gfCNCPoint2[10772] = {X 54.3258, Y 60.4704, Z -3.0000, A 0.000, B 0.000, C 0.000 }
gfCNCPoint2[10773] = {X 52.7011, Y 61.0822, Z -3.0000, A 0.000, B 0.000, C 0.000 }
gfCNCPoint2[10774] = {X 51.0221, Y 61.5238, Z -3.0000, A 0.000, B 0.000, C 0.000 }
gfCNCPoint2[10775] = {X 49.3067, Y 61.7907, Z -3.0000, A 0.000, B 0.000, C 0.000 }
gfCNCPoint2[10776] = {X 47.5729, Y 61.8800, Z -3.0000, A 0.000, B 0.000, C 0.000 }
gfCNCPoint2[10777] = {X 40.6393, Y 61.8800, Z -3.0000, A 0.000, B 0.000, C 0.000 }
gfCNCPoint2[10778] = {X 39.0676, Y 61.8067, Z -3.0000, A 0.000, B 0.000, C 0.000 }
gfCNCPoint2[10779] = {X 37.5096, Y 61.5873, Z -3.0000, A 0.000, B 0.000, C 0.000 }
gfCNCPoint2[10780] = {X 35.9787, Y 61.2239, Z -3.0000, A 0.000, B 0.000, C 0.000 }
gfCNCPoint2[10781] = {X 34.3400, Y 61.9594, Z -3.0000, A 0.000, B 0.000, C 0.000 }
gfCNCPoint2[10782] = {X 32.6450, Y 62.5538, Z -3.0000, A 0.000, B 0.000, C 0.000 }
gfCNCPoint2[10783] = {X 30.9057, Y 63.0026, Z -3.0000, A 0.000, B 0.000, C 0.000 }
gfCNCPoint2[10784] = {X 29.1347, Y 63.3027, Z -3.0000, A 0.000, B 0.000, C 0.000 }
gfCNCPoint2[10785] = {X 27.5576, Y 63.9540, Z -3.0000, A 0.000, B 0.000, C 0.000 }
gfCNCPoint2[10786] = {X 25.9568, Y 64.5448, Z -3.0000, A 0.000, B 0.000, C 0.000 }
gfCNCPoint2[10787] = {X 23.6955, Y 65.2843, Z -3.0000, A 0.000, B 0.000, C 0.000 }
gfCNCPoint2[10788] = {X 21.3940, Y 65.8871, Z -3.0000, A 0.000, B 0.000, C 0.000 }
gfCNCPoint2[10789] = {X 19.0606, Y 66.3509, Z -3.0000, A 0.000, B 0.000, C 0.000 }
gfCNCPoint2[10790] = {X 16.7035, Y 66.6740, Z -3.0000, A 0.000, B 0.000, C 0.000 }
gfCNCPoint2[10791] = {X 16.7035, Y 83.2950, Z -3.0000, A 0.000, B 0.000, C 0.000 }
gfCNCPoint2[10792] = {X 111.5064, Y 83.2950, Z -3.0000, A 0.000, B 0.000, C 0.000 }
gfCNCPoint2[10793] = {X 113.0153, Y 81.9635, Z -3.0000, A 0.000, B 0.000, C 0.000 }
gfCNCPoint2[10794] = {X 114.6547, Y 80.7965, Z -3.0000, A 0.000, B 0.000, C 0.000 }
gfCNCPoint2[10795] = {X 116.4069, Y 79.8068, Z -3.0000, A 0.000, B 0.000, C 0.000 }
gfCNCPoint2[10796] = {X 117.4766, Y 81.9553, Z -3.0000, A 0.000, B 0.000, C 0.000 }
gfCNCPoint2[10797] = {X 119.1631, Y 81.2272, Z -3.0000, A 0.000, B 0.000, C 0.000 }
gfCNCPoint2[10798] = {X 120.9187, Y 80.6868, Z -3.0000, A 0.000, B 0.000, C 0.000 }
gfCNCPoint2[10799] = {X 142.4298, Y 57.0646, Z -3.0000, A 0.000, B 0.000, C 0.000 }
gfCNCPoint2[10800] = {X 141.1668, Y 56.9339, Z -3.0000, A 0.000, B 0.000, C 0.000 }
gfCNCPoint2[10801] = {X 139.9244, Y 56.6714, Z -3.0000, A 0.000, B 0.000, C 0.000 }
gfCNCPoint2[10802] = {X 138.7165, Y 56.2799, Z -3.0000, A 0.000, B 0.000, C 0.000 }
gfCNCPoint2[10803] = {X 137.2794, Y 55.6182, Z -3.0000, A 0.000, B 0.000, C 0.000 }
gfCNCPoint2[10804] = {X 135.9410, Y 54.7743, Z -3.0000, A 0.000, B 0.000, C 0.000 }
gfCNCPoint2[10805] = {X 134.7245, Y 53.7627, Z -3.0000, A 0.000, B 0.000, C 0.000 }
gfCNCPoint2[10806] = {X 133.6506, Y 52.6008, Z -3.0000, A 0.000, B 0.000, C 0.000 }
gfCNCPoint2[10807] = {X 132.7377, Y 51.3086, Z -3.0000, A 0.000, B 0.000, C 0.000 }
gfCNCPoint2[10808] = {X 132.0016, Y 49.9081, Z -3.0000, A 0.000, B 0.000, C 0.000 }
gfCNCPoint2[10809] = {X 131.4549, Y 48.4234, Z -3.0000, A 0.000, B 0.000, C 0.000 }
gfCNCPoint2[10810] = {X 131.1845, Y 47.3200, Z -3.0000, A 0.000, B 0.000, C 0.000 }
gfCNCPoint2[10811] = {X 131.0190, Y 46.1961, Z -3.0000, A 0.000, B 0.000, C 0.000 }
gfCNCPoint2[10812] = {X 130.9598, Y 45.0616, Z -3.0000, A 0.000, B 0.000, C 0.000 }
gfCNCPoint2[10813] = {X 130.9601, Y 44.0979, Z -3.0000, A 0.000, B 0.000, C 0.000 }
gfCNCPoint2[10814] = {X 131.0921, Y 42.4244, Z -3.0000, A 0.000, B 0.000, C 0.000 }
gfCNCPoint2[10815] = {X 131.4548, Y 40.7854, Z -3.0000, A 0.000, B 0.000, C 0.000 }
gfCNCPoint2[10816] = {X 133.7565, Y 41.4655, Z -3.0000, A 0.000, B 0.000, C 0.000 }
gfCNCPoint2[10817] = {X 134.2330, Y 40.1906, Z -3.0000, A 0.000, B 0.000, C 0.000 }
gfCNCPoint2[10818] = {X 134.8836, Y 38.9952, Z -3.0000, A 0.000, B 0.000, C 0.000 }
gfCNCPoint2[10819] = {X 134.8836, Y 27.0854, Z -3.0000, A 0.000, B 0.000, C 0.000 }
gfCNCPoint2[10820] = {X 134.3931, Y 27.1259, Z -3.0000, A 0.000, B 0.000, C 0.000 }
gfCNCPoint2[10821] = {X 133.9011, Y 27.1414, Z -3.0000, A 0.000, B 0.000, C 0.000 }
gfCNCPoint2[10822] = {X 133.2006, Y 27.1415, Z -3.0000, A 0.000, B 0.000, C 0.000 }
gfCNCPoint2[10823] = {X 131.9566, Y 27.0613, Z -3.0000, A 0.000, B 0.000, C 0.000 }
gfCNCPoint2[10824] = {X 130.7331, Y 26.8218, Z -3.0000, A 0.000, B 0.000, C 0.000 }
gfCNCPoint2[10825] = {X 129.5506, Y 26.4270, Z -3.0000, A 0.000, B 0.000, C 0.000 }
gfCNCPoint2[10826] = {X 128.4287, Y 25.8836, Z -3.0000, A 0.000, B 0.000, C 0.000 }
gfCNCPoint2[10827] = {X 127.3858, Y 25.2004, Z -3.0000, A 0.000, B 0.000, C 0.000 }
gfCNCPoint2[10828] = {X 126.3445, Y 24.2950, Z -3.0000, A 0.000, B 0.000, C 0.000 }
gfCNCPoint2[10829] = {X 125.4425, Y 23.2506, Z -3.0000, A 0.000, B 0.000, C 0.000 }
gfCNCPoint2[10830] = {X 124.6982, Y 22.0887, Z -3.0000, A 0.000, B 0.000, C 0.000 }
gfCNCPoint2[10831] = {X 124.1266, Y 20.8327, Z -3.0000, A 0.000, B 0.000, C 0.000 }
gfCNCPoint2[10832] = {X 123.7395, Y 19.5081, Z -3.0000, A 0.000, B 0.000, C 0.000 }
gfCNCPoint2[10833] = {X 123.5446, Y 18.1420, Z -3.0000, A 0.000, B 0.000, C 0.000 }
gfCNCPoint2[10834] = {X 123.5435, Y 39.7463, Z -3.0000, A 0.000, B 0.000, C 0.000 }
gfCNCPoint2[10835] = {X 124.1923, Y 40.7404, Z -3.0000, A 0.000, B 0.000, C 0.000 }
gfCNCPoint2[10836] = {X 124.6708, Y 41.8267, Z -3.0000, A 0.000, B 0.000, C 0.000 }
gfCNCPoint2[10837] = {X 124.9665, Y 42.9763, Z -3.0000, A 0.000, B 0.000, C 0.000 }
gfCNCPoint2[10838] = {X 125.0714, Y 44.1587, Z -3.0000, A 0.000, B 0.000, C 0.000 }
gfCNCPoint2[10839] = {X 125.0716, Y 45.0000, Z -3.0000, A 0.000, B 0.000, C 0.000 }
gfCNCPoint2[10840] = {X 124.9610, Y 46.2642, Z -3.0000, A 0.000, B 0.000, C 0.000 }
gfCNCPoint2[10841] = {X 124.6325, Y 47.4899, Z -3.0000, A 0.000, B 0.000, C 0.000 }
gfCNCPoint2[10842] = {X 124.0962, Y 48.6400, Z -3.0000, A 0.000, B 0.000, C 0.000 }
gfCNCPoint2[10843] = {X 123.3684, Y 49.6795, Z -3.0000, A 0.000, B 0.000, C 0.000 }
gfCNCPoint2[10844] = {X 122.4711, Y 50.5768, Z -3.0000, A 0.000, B 0.000, C 0.000 }
gfCNCPoint2[10845] = {X 121.4316, Y 51.3047, Z -3.0000, A 0.000, B 0.000, C 0.000 }
gfCNCPoint2[10846] = {X 120.2815, Y 51.8410, Z -3.0000, A 0.000, B 0.000, C 0.000 }
gfCNCPoint2[10847] = {X 119.0557, Y 52.1694, Z -3.0000, A 0.000, B 0.000, C 0.000 }
gfCNCPoint2[10848] = {X 117.7916, Y 52.2800, Z -3.0000, A 0.000, B 0.000, C 0.000 }
gfCNCPoint2[10849] = {X 111.9185, Y 52.2800, Z -3.0000, A 0.000, B 0.000, C 0.000 }
gfCNCPoint2[10850] = {X 110.8481, Y 52.2009, Z -3.0000, A 0.000, B 0.000, C 0.000 }
gfCNCPoint2[10851] = {X 109.8009, Y 51.9652, Z -3.0000, A 0.000, B 0.000, C 0.000 }
gfCNCPoint2[10852] = {X 108.7998, Y 51.5782, Z -3.0000, A 0.000, B 0.000, C 0.000 }
gfCNCPoint2[10853] = {X 107.8665, Y 51.0481, Z -3.0000, A 0.000, B 0.000, C 0.000 }
gfCNCPoint2[10854] = {X 107.0213, Y 50.3866, Z -3.0000, A 0.000, B 0.000, C 0.000 }
gfCNCPoint2[10855] = {X 106.1743, Y 51.0493, Z -3.0000, A 0.000, B 0.000, C 0.000 }
gfCNCPoint2[10856] = {X 105.2389, Y 51.5800, Z -3.0000, A 0.000, B 0.000, C 0.000 }
gfCNCPoint2[10857] = {X 104.0917, Y 52.0091, Z -3.0000, A 0.000, B 0.000, C 0.000 }
